KUKA KRL program: part3_2_post.src

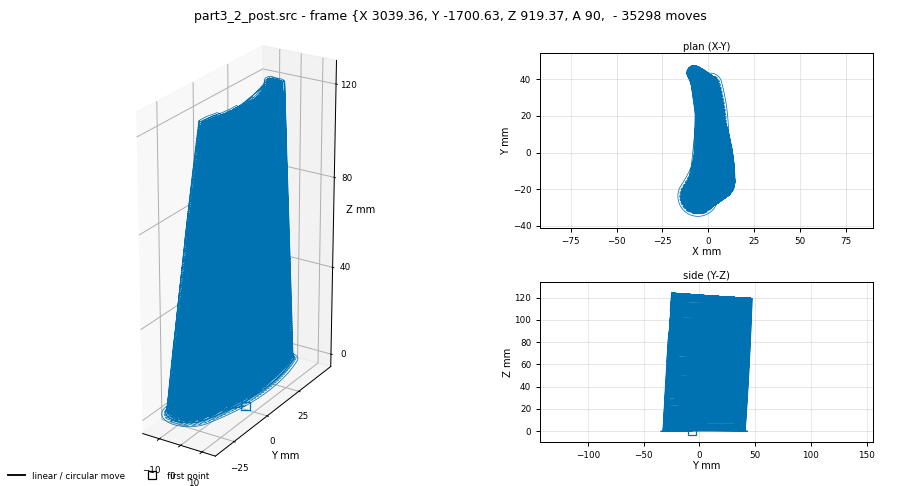
[picture p0: tool path of part3_2_post.src in frame {X 3039.36, Y -1700.63, Z 919.37, A 90, , 35298 of 35299 moves have a stored position in this frame; points joined in program order, loops and branches not executed]
&ACCESS RVO
&REL 3
DEF part3_2_post ( )

   ;---------------------RSI variable--------------------
   ; Declaration of KRL variables
   DECL INT ret	; Return value for RSI commands
   DECL INT CONTID	; ContainerID
   ;---------------------RSI variable--------------------

   ;---------------------RSI --------------------
   ret = RSI_CREATE("ros_rsi",CONTID,TRUE)
   IF (ret <> RSIOK) THEN
      HALT
   ENDIF

   ; Start RSI execution
   ret = RSI_ON(#ABSOLUTE)
   IF (ret <> RSIOK) THEN
      HALT
   ENDIF
   ;---------------------RSI--------------------

   ;FOLD INI
      ;FOLD BASISTECH INI
         GLOBAL INTERRUPT DECL 3 WHEN $STOPMESS==TRUE DO IR_STOPM ( )
         INTERRUPT ON 3
         BAS (#INITMOV,0 )
      ;ENDFOLD (BASISTECH INI)
      ;FOLD USER INI
         ;Make your modifications here

      ;ENDFOLD (USER INI)
   ;ENDFOLD (INI)

   $TOOL=TOOL_DATA[1] ; "LASER"
   ;$TOOL={X -5.25,Y -259.33,Z 286.75,A 0.0,B 0.0,C 0.0}
   $BASE={X 3039.36, Y -1700.63, Z 919.37, A 90, B 0, C 0}  ; user-defined BASE frame
   ;$BASE=BASE_DATA[3] ; user-defined BASE frame
   ;$BASE=BASE_DATA[1] ; "LK_BASE (TurnTable)"
   ;$BASE={X 1622.85,Y -1582.69,Z 15.62,A 0.14,B 0.07,C 0.25}

   $VEL.CP = 0.020 ; linear speed m/s
   $VEL.ORI1 = 300 ; swivel speed deg/s
   $VEL.ORI2 = 300 ; rotation speed deg/s

   $APO.CDIS = 0.3 ;mm; in ABB: zonddata = z0

   PTP $POS_ACT
   $OUT[15]=TRUE ; Wire touch signal bypass
   LaserOn_Ext()

   ;FOLD ANOUT ql_Power=0.1 ;%{PE}%R 8.5.19,%MKUKATPBASIS,%CANA,%VANOUT_STAT,%P 2:CHANNEL_1, 4:0.1
      $ANOUT[1]=0.179
   ;ENDFOLD

   LIN {X 9.999, Y -6.495, Z 0.000}
   LaserStart_Ext()
   LIN {X 9.851, Y -7.487, Z 0.000} C_DIS
   LIN {X 9.694, Y -8.478, Z 0.000} C_DIS
   LIN {X 9.517, Y -9.533, Z 0.000} C_DIS
   LIN {X 9.342, Y -10.520, Z 0.000} C_DIS
   LIN {X 9.158, Y -11.507, Z 0.000} C_DIS
   LIN {X 8.966, Y -12.491, Z 0.000} C_DIS
   LIN {X 8.778, Y -13.409, Z 0.000} C_DIS
   LIN {X 8.568, Y -14.390, Z 0.000} C_DIS
   LIN {X 8.350, Y -15.371, Z 0.000} C_DIS
   LIN {X 8.122, Y -16.349, Z 0.000} C_DIS
   LIN {X 7.886, Y -17.327, Z 0.000} C_DIS
   LIN {X 7.641, Y -18.302, Z 0.000} C_DIS
   LIN {X 7.387, Y -19.277, Z 0.000} C_DIS
   LIN {X 7.124, Y -20.250, Z 0.000} C_DIS
   LIN {X 6.851, Y -21.221, Z 0.000} C_DIS
   LIN {X 6.570, Y -22.190, Z 0.000} C_DIS
   LIN {X 6.300, Y -23.094, Z 0.000} C_DIS
   LIN {X 6.001, Y -24.061, Z 0.000} C_DIS
   LIN {X 5.693, Y -25.026, Z 0.000} C_DIS
   LIN {X 5.397, Y -25.926, Z 0.000} C_DIS
   LIN {X 5.181, Y -26.567, Z 0.000} C_DIS
   LIN {X 5.050, Y -26.952, Z 0.000} C_DIS
   LIN {X 4.961, Y -27.208, Z 0.000} C_DIS
   LIN {X 4.917, Y -27.337, Z 0.000} C_DIS
   LIN {X 4.841, Y -27.550, Z 0.000} C_DIS
   LIN {X 4.691, Y -27.934, Z 0.000} C_DIS
   LIN {X 4.448, Y -28.479, Z 0.000} C_DIS
   LIN {X 4.032, Y -29.267, Z 0.000} C_DIS
   LIN {X 3.511, Y -30.081, Z 0.000} C_DIS
   LIN {X 2.916, Y -30.853, Z 0.000} C_DIS
   LIN {X 2.255, Y -31.570, Z 0.000} C_DIS
   LIN {X 1.511, Y -32.247, Z 0.000} C_DIS
   LIN {X 0.738, Y -32.833, Z 0.000} C_DIS
   LIN {X -0.089, Y -33.352, Z 0.000} C_DIS
   LIN {X -0.956, Y -33.796, Z 0.000} C_DIS
   LIN {X -1.890, Y -34.172, Z 0.000} C_DIS
   LIN {X -2.855, Y -34.463, Z 0.000} C_DIS
   LIN {X -3.812, Y -34.661, Z 0.000} C_DIS
   LIN {X -4.777, Y -34.773, Z 0.000} C_DIS
   LIN {X -5.745, Y -34.799, Z 0.000} C_DIS
   LIN {X -6.715, Y -34.739, Z 0.000} C_DIS
   LIN {X -7.682, Y -34.593, Z 0.000} C_DIS
   LIN {X -8.661, Y -34.354, Z 0.000} C_DIS
   LIN {X -9.578, Y -34.041, Z 0.000} C_DIS
   LIN {X -10.468, Y -33.646, Z 0.000} C_DIS
   LIN {X -11.321, Y -33.170, Z 0.000} C_DIS
   LIN {X -12.123, Y -32.625, Z 0.000} C_DIS
   LIN {X -12.873, Y -32.012, Z 0.000} C_DIS
   LIN {X -13.571, Y -31.330, Z 0.000} C_DIS
   LIN {X -14.205, Y -30.589, Z 0.000} C_DIS
   LIN {X -14.787, Y -29.768, Z 0.000} C_DIS
   LIN {X -15.273, Y -28.929, Z 0.000} C_DIS
   LIN {X -15.686, Y -28.043, Z 0.000} C_DIS
   LIN {X -16.017, Y -27.128, Z 0.000} C_DIS
   LIN {X -16.282, Y -26.120, Z 0.000} C_DIS
   LIN {X -16.440, Y -25.161, Z 0.000} C_DIS
   LIN {X -16.513, Y -24.186, Z 0.000} C_DIS
   LIN {X -16.499, Y -23.215, Z 0.000} C_DIS
   LIN {X -16.400, Y -22.252, Z 0.000} C_DIS
   LIN {X -16.208, Y -21.260, Z 0.000} C_DIS
   LIN {X -15.937, Y -20.321, Z 0.000} C_DIS
   LIN {X -15.586, Y -19.416, Z 0.000} C_DIS
   LIN {X -15.139, Y -18.514, Z 0.000} C_DIS
   LIN {X -14.672, Y -17.743, Z 0.000} C_DIS
   LIN {X -14.112, Y -16.887, Z 0.000} C_DIS
   LIN {X -13.565, Y -16.024, Z 0.000} C_DIS
   LIN {X -13.060, Y -15.203, Z 0.000} C_DIS
   LIN {X -12.510, Y -14.277, Z 0.000} C_DIS
   LIN {X -12.002, Y -13.394, Z 0.000} C_DIS
   LIN {X -11.507, Y -12.503, Z 0.000} C_DIS
   LIN {X -11.025, Y -11.607, Z 0.000} C_DIS
   LIN {X -10.583, Y -10.753, Z 0.000} C_DIS
   LIN {X -10.126, Y -9.842, Z 0.000} C_DIS
   LIN {X -9.707, Y -8.975, Z 0.000} C_DIS
   LIN {X -9.276, Y -8.052, Z 0.000} C_DIS
   LIN {X -8.858, Y -7.124, Z 0.000} C_DIS
   LIN {X -8.455, Y -6.192, Z 0.000} C_DIS
   LIN {X -8.067, Y -5.258, Z 0.000} C_DIS
   LIN {X -7.693, Y -4.321, Z 0.000} C_DIS
   LIN {X -7.353, Y -3.432, Z 0.000} C_DIS
   LIN {X -6.987, Y -2.433, Z 0.000} C_DIS
   LIN {X -6.654, Y -1.483, Z 0.000} C_DIS
   LIN {X -6.352, Y -0.580, Z 0.000} C_DIS
   LIN {X -6.028, Y 0.435, Z 0.000} C_DIS
   LIN {X -5.735, Y 1.402, Z 0.000} C_DIS
   LIN {X -5.456, Y 2.373, Z 0.000} C_DIS
   LIN {X -5.163, Y 3.454, Z 0.000} C_DIS
   LIN {X -4.928, Y 4.375, Z 0.000} C_DIS
   LIN {X -4.693, Y 5.354, Z 0.000} C_DIS
   LIN {X -4.472, Y 6.338, Z 0.000} C_DIS
   LIN {X -4.264, Y 7.327, Z 0.000} C_DIS
   LIN {X -4.080, Y 8.268, Z 0.000} C_DIS
   LIN {X -3.900, Y 9.268, Z 0.000} C_DIS
   LIN {X -3.742, Y 10.214, Z 0.000} C_DIS
   LIN {X -3.582, Y 11.276, Z 0.000} C_DIS
   LIN {X -3.452, Y 12.228, Z 0.000} C_DIS
   LIN {X -3.328, Y 13.242, Z 0.000} C_DIS
   LIN {X -3.225, Y 14.200, Z 0.000} C_DIS
   LIN {X -3.130, Y 15.210, Z 0.000} C_DIS
   LIN {X -3.051, Y 16.218, Z 0.000} C_DIS
   LIN {X -2.988, Y 17.171, Z 0.000} C_DIS
   LIN {X -2.937, Y 18.180, Z 0.000} C_DIS
   LIN {X -2.899, Y 19.191, Z 0.000} C_DIS
   LIN {X -2.877, Y 20.145, Z 0.000} C_DIS
   LIN {X -2.868, Y 21.157, Z 0.000} C_DIS
   LIN {X -2.873, Y 22.168, Z 0.000} C_DIS
   LIN {X -2.891, Y 23.123, Z 0.000} C_DIS
   LIN {X -2.924, Y 24.133, Z 0.000} C_DIS
   LIN {X -2.971, Y 25.142, Z 0.000} C_DIS
   LIN {X -3.029, Y 26.094, Z 0.000} C_DIS
   LIN {X -3.104, Y 27.100, Z 0.000} C_DIS
   LIN {X -3.194, Y 28.106, Z 0.000} C_DIS
   LIN {X -3.291, Y 29.054, Z 0.000} C_DIS
   LIN {X -3.408, Y 30.058, Z 0.000} C_DIS
   LIN {X -3.540, Y 31.060, Z 0.000} C_DIS
   LIN {X -3.694, Y 32.116, Z 0.000} C_DIS
   LIN {X -3.855, Y 33.116, Z 0.000} C_DIS
   LIN {X -4.030, Y 34.115, Z 0.000} C_DIS
   LIN {X -4.219, Y 35.112, Z 0.000} C_DIS
   LIN {X -4.423, Y 36.108, Z 0.000} C_DIS
   LIN {X -4.573, Y 37.126, Z 0.000} C_DIS
   LIN {X -4.539, Y 38.127, Z 0.000} C_DIS
   LIN {X -4.338, Y 39.115, Z 0.000} C_DIS
   LIN {X -3.977, Y 40.053, Z 0.000} C_DIS
   LIN {X -3.442, Y 40.941, Z 0.000} C_DIS
   LIN {X -2.768, Y 41.711, Z 0.000} C_DIS
   LIN {X -1.943, Y 42.381, Z 0.000} C_DIS
   LIN {X -1.067, Y 42.875, Z 0.000} C_DIS
   LIN {X -0.126, Y 43.212, Z 0.000} C_DIS
   LIN {X 0.876, Y 43.381, Z 0.000} C_DIS
   LIN {X 1.877, Y 43.376, Z 0.000} C_DIS
   LIN {X 2.884, Y 43.202, Z 0.000} C_DIS
   LIN {X 3.835, Y 42.872, Z 0.000} C_DIS
   LIN {X 4.720, Y 42.387, Z 0.000} C_DIS
   LIN {X 5.506, Y 41.764, Z 0.000} C_DIS
   LIN {X 6.189, Y 41.003, Z 0.000} C_DIS
   LIN {X 6.758, Y 40.100, Z 0.000} C_DIS
   LIN {X 7.051, Y 39.435, Z 0.000} C_DIS
   LIN {X 7.216, Y 38.908, Z 0.000} C_DIS
   LIN {X 7.443, Y 38.057, Z 0.000} C_DIS
   LIN {X 7.697, Y 37.073, Z 0.000} C_DIS
   LIN {X 7.926, Y 36.154, Z 0.000} C_DIS
   LIN {X 8.177, Y 35.103, Z 0.000} C_DIS
   LIN {X 8.404, Y 34.115, Z 0.000} C_DIS
   LIN {X 8.621, Y 33.127, Z 0.000} C_DIS
   LIN {X 8.816, Y 32.203, Z 0.000} C_DIS
   LIN {X 9.042, Y 31.080, Z 0.000} C_DIS
   LIN {X 9.232, Y 30.088, Z 0.000} C_DIS
   LIN {X 9.413, Y 29.095, Z 0.000} C_DIS
   LIN {X 9.585, Y 28.100, Z 0.000} C_DIS
   LIN {X 9.738, Y 27.171, Z 0.000} C_DIS
   LIN {X 9.892, Y 26.174, Z 0.000} C_DIS
   LIN {X 10.038, Y 25.176, Z 0.000} C_DIS
   LIN {X 10.174, Y 24.176, Z 0.000} C_DIS
   LIN {X 10.294, Y 23.242, Z 0.000} C_DIS
   LIN {X 10.414, Y 22.241, Z 0.000} C_DIS
   LIN {X 10.531, Y 21.171, Z 0.000} C_DIS
   LIN {X 10.626, Y 20.234, Z 0.000} C_DIS
   LIN {X 10.718, Y 19.228, Z 0.000} C_DIS
   LIN {X 10.802, Y 18.222, Z 0.000} C_DIS
   LIN {X 10.872, Y 17.281, Z 0.000} C_DIS
   LIN {X 10.938, Y 16.273, Z 0.000} C_DIS
   LIN {X 10.995, Y 15.262, Z 0.000} C_DIS
   LIN {X 11.043, Y 14.251, Z 0.000} C_DIS
   LIN {X 11.080, Y 13.306, Z 0.000} C_DIS
   LIN {X 11.110, Y 12.292, Z 0.000} C_DIS
   LIN {X 11.131, Y 11.277, Z 0.000} C_DIS
   LIN {X 11.143, Y 10.328, Z 0.000} C_DIS
   LIN {X 11.146, Y 9.313, Z 0.000} C_DIS
   LIN {X 11.141, Y 8.365, Z 0.000} C_DIS
   LIN {X 11.126, Y 7.350, Z 0.000} C_DIS
   LIN {X 11.103, Y 6.336, Z 0.000} C_DIS
   LIN {X 11.070, Y 5.325, Z 0.000} C_DIS
   LIN {X 11.031, Y 4.382, Z 0.000} C_DIS
   LIN {X 10.980, Y 3.374, Z 0.000} C_DIS
   LIN {X 10.921, Y 2.367, Z 0.000} C_DIS
   LIN {X 10.852, Y 1.361, Z 0.000} C_DIS
   LIN {X 10.774, Y 0.358, Z 0.000} C_DIS
   LIN {X 10.694, Y -0.578, Z 0.000} C_DIS
   LIN {X 10.599, Y -1.579, Z 0.000} C_DIS
   LIN {X 10.495, Y -2.578, Z 0.000} C_DIS
   LIN {X 10.382, Y -3.576, Z 0.000} C_DIS
   LIN {X 10.260, Y -4.573, Z 0.000} C_DIS
   LIN {X 10.138, Y -5.502, Z 0.000} C_DIS
   LIN {X 9.999, Y -6.495, Z 0.000}
   LaserEnd_Ext()
   LIN {X -8.478, Y -33.360, Z 0.000}
   LaserStart_Ext()
   LIN {X -2.661, Y -33.360, Z 0.000}
   LaserEnd_Ext()
   LIN {X -0.389, Y -32.360, Z 0.000}
   LaserStart_Ext()
   LIN {X -10.721, Y -32.360, Z 0.000}
   LaserEnd_Ext()
   LIN {X -12.090, Y -31.360, Z 0.000}
   LaserStart_Ext()
   LIN {X 1.000, Y -31.360, Z 0.000}
   LaserEnd_Ext()
   LIN {X 2.010, Y -30.360, Z 0.000}
   LaserStart_Ext()
   LIN {X -13.085, Y -30.360, Z 0.000}
   LaserEnd_Ext()
   LIN {X -13.850, Y -29.360, Z 0.000}
   LaserStart_Ext()
   LIN {X 2.785, Y -29.360, Z 0.000}
   LaserEnd_Ext()
   LIN {X 3.380, Y -28.360, Z 0.000}
   LaserStart_Ext()
   LIN {X -14.435, Y -28.360, Z 0.000}
   LaserEnd_Ext()
   LIN {X -14.870, Y -27.360, Z 0.000}
   LaserStart_Ext()
   LIN {X 3.841, Y -27.360, Z 0.000}
   LaserEnd_Ext()
   LIN {X 4.196, Y -26.360, Z 0.000}
   LaserStart_Ext()
   LIN {X -15.185, Y -26.360, Z 0.000}
   LaserEnd_Ext()
   LIN {X -15.394, Y -25.360, Z 0.000}
   LaserStart_Ext()
   LIN {X 4.531, Y -25.360, Z 0.000}
   LaserEnd_Ext()
   LIN {X 4.856, Y -24.360, Z 0.000}
   LaserStart_Ext()
   LIN {X -15.497, Y -24.360, Z 0.000}
   LaserEnd_Ext()
   LIN {X -15.501, Y -23.360, Z 0.000}
   LaserStart_Ext()
   LIN {X 5.171, Y -23.360, Z 0.000}
   LaserEnd_Ext()
   LIN {X 5.475, Y -22.360, Z 0.000}
   LaserStart_Ext()
   LIN {X -15.403, Y -22.360, Z 0.000}
   LaserEnd_Ext()
   LIN {X -15.196, Y -21.360, Z 0.000}
   LaserStart_Ext()
   LIN {X 5.770, Y -21.360, Z 0.000}
   LaserEnd_Ext()
   LIN {X 6.054, Y -20.360, Z 0.000}
   LaserStart_Ext()
   LIN {X -14.879, Y -20.360, Z 0.000}
   LaserEnd_Ext()
   LIN {X -14.442, Y -19.360, Z 0.000}
   LaserStart_Ext()
   LIN {X 6.328, Y -19.360, Z 0.000}
   LaserEnd_Ext()
   LIN {X 6.592, Y -18.360, Z 0.000}
   LaserStart_Ext()
   LIN {X -13.876, Y -18.360, Z 0.000}
   LaserEnd_Ext()
   LIN {X -13.228, Y -17.360, Z 0.000}
   LaserStart_Ext()
   LIN {X 6.847, Y -17.360, Z 0.000}
   LaserEnd_Ext()
   LIN {X 7.091, Y -16.360, Z 0.000}
   LaserStart_Ext()
   LIN {X -12.598, Y -16.360, Z 0.000}
   LaserEnd_Ext()
   LIN {X -11.990, Y -15.360, Z 0.000}
   LaserStart_Ext()
   LIN {X 7.326, Y -15.360, Z 0.000}
   LaserEnd_Ext()
   LIN {X 7.551, Y -14.360, Z 0.000}
   LaserStart_Ext()
   LIN {X -11.404, Y -14.360, Z 0.000}
   LaserEnd_Ext()
   LIN {X -10.839, Y -13.360, Z 0.000}
   LaserStart_Ext()
   LIN {X 7.766, Y -13.360, Z 0.000}
   LaserEnd_Ext()
   LIN {X 7.972, Y -12.360, Z 0.000}
   LaserStart_Ext()
   LIN {X -10.295, Y -12.360, Z 0.000}
   LaserEnd_Ext()
   LIN {X -9.771, Y -11.360, Z 0.000}
   LaserStart_Ext()
   LIN {X 8.168, Y -11.360, Z 0.000}
   LaserEnd_Ext()
   LIN {X 8.355, Y -10.360, Z 0.000}
   LaserStart_Ext()
   LIN {X -9.267, Y -10.360, Z 0.000}
   LaserEnd_Ext()
   LIN {X -8.783, Y -9.360, Z 0.000}
   LaserStart_Ext()
   LIN {X 8.532, Y -9.360, Z 0.000}
   LaserEnd_Ext()
   LIN {X 8.700, Y -8.360, Z 0.000}
   LaserStart_Ext()
   LIN {X -8.318, Y -8.360, Z 0.000}
   LaserEnd_Ext()
   LIN {X -7.871, Y -7.360, Z 0.000}
   LaserStart_Ext()
   LIN {X 8.859, Y -7.360, Z 0.000}
   LaserEnd_Ext()
   LIN {X 9.008, Y -6.360, Z 0.000}
   LaserStart_Ext()
   LIN {X -7.442, Y -6.360, Z 0.000}
   LaserEnd_Ext()
   LIN {X -7.031, Y -5.360, Z 0.000}
   LaserStart_Ext()
   LIN {X 9.148, Y -5.360, Z 0.000}
   LaserEnd_Ext()
   LIN {X 9.278, Y -4.360, Z 0.000}
   LaserStart_Ext()
   LIN {X -6.638, Y -4.360, Z 0.000}
   LaserEnd_Ext()
   LIN {X -6.261, Y -3.360, Z 0.000}
   LaserStart_Ext()
   LIN {X 9.400, Y -3.360, Z 0.000}
   LaserEnd_Ext()
   LIN {X 9.512, Y -2.360, Z 0.000}
   LaserStart_Ext()
   LIN {X -5.902, Y -2.360, Z 0.000}
   LaserEnd_Ext()
   LIN {X -5.558, Y -1.360, Z 0.000}
   LaserStart_Ext()
   LIN {X 9.615, Y -1.360, Z 0.000}
   LaserEnd_Ext()
   LIN {X 9.709, Y -0.360, Z 0.000}
   LaserStart_Ext()
   LIN {X -5.232, Y -0.360, Z 0.000}
   LaserEnd_Ext()
   LIN {X -4.921, Y 0.640, Z 0.000}
   LaserStart_Ext()
   LIN {X 9.793, Y 0.640, Z 0.000}
   LaserEnd_Ext()
   LIN {X 9.869, Y 1.640, Z 0.000}
   LaserStart_Ext()
   LIN {X -4.627, Y 1.640, Z 0.000}
   LaserEnd_Ext()
   LIN {X -4.348, Y 2.640, Z 0.000}
   LaserStart_Ext()
   LIN {X 9.935, Y 2.640, Z 0.000}
   LaserEnd_Ext()
   LIN {X 9.992, Y 3.640, Z 0.000}
   LaserStart_Ext()
   LIN {X -4.084, Y 3.640, Z 0.000}
   LaserEnd_Ext()
   LIN {X -3.836, Y 4.640, Z 0.000}
   LaserStart_Ext()
   LIN {X 10.041, Y 4.640, Z 0.000}
   LaserEnd_Ext()
   LIN {X 10.080, Y 5.640, Z 0.000}
   LaserStart_Ext()
   LIN {X -3.604, Y 5.640, Z 0.000}
   LaserEnd_Ext()
   LIN {X -3.387, Y 6.640, Z 0.000}
   LaserStart_Ext()
   LIN {X 10.110, Y 6.640, Z 0.000}
   LaserEnd_Ext()
   LIN {X 10.130, Y 7.640, Z 0.000}
   LaserStart_Ext()
   LIN {X -3.184, Y 7.640, Z 0.000}
   LaserEnd_Ext()
   LIN {X -2.997, Y 8.640, Z 0.000}
   LaserStart_Ext()
   LIN {X 10.142, Y 8.640, Z 0.000}
   LaserEnd_Ext()
   LIN {X 10.145, Y 9.640, Z 0.000}
   LaserStart_Ext()
   LIN {X -2.824, Y 9.640, Z 0.000}
   LaserEnd_Ext()
   LIN {X -2.667, Y 10.640, Z 0.000}
   LaserStart_Ext()
   LIN {X 10.139, Y 10.640, Z 0.000}
   LaserEnd_Ext()
   LIN {X 10.123, Y 11.640, Z 0.000}
   LaserStart_Ext()
   LIN {X -2.523, Y 11.640, Z 0.000}
   LaserEnd_Ext()
   LIN {X -2.394, Y 12.640, Z 0.000}
   LaserStart_Ext()
   LIN {X 10.099, Y 12.640, Z 0.000}
   LaserEnd_Ext()
   LIN {X 10.066, Y 13.640, Z 0.000}
   LaserStart_Ext()
   LIN {X -2.280, Y 13.640, Z 0.000}
   LaserEnd_Ext()
   LIN {X -2.179, Y 14.640, Z 0.000}
   LaserStart_Ext()
   LIN {X 10.024, Y 14.640, Z 0.000}
   LaserEnd_Ext()
   LIN {X 9.972, Y 15.640, Z 0.000}
   LaserStart_Ext()
   LIN {X -2.093, Y 15.640, Z 0.000}
   LaserEnd_Ext()
   LIN {X -2.021, Y 16.640, Z 0.000}
   LaserStart_Ext()
   LIN {X 9.912, Y 16.640, Z 0.000}
   LaserEnd_Ext()
   LIN {X 9.842, Y 17.640, Z 0.000}
   LaserStart_Ext()
   LIN {X -1.963, Y 17.640, Z 0.000}
   LaserEnd_Ext()
   LIN {X -1.919, Y 18.640, Z 0.000}
   LaserStart_Ext()
   LIN {X 9.764, Y 18.640, Z 0.000}
   LaserEnd_Ext()
   LIN {X 9.676, Y 19.640, Z 0.000}
   LaserStart_Ext()
   LIN {X -1.889, Y 19.640, Z 0.000}
   LaserEnd_Ext()
   LIN {X -1.873, Y 20.640, Z 0.000}
   LaserStart_Ext()
   LIN {X 9.580, Y 20.640, Z 0.000}
   LaserEnd_Ext()
   LIN {X 9.474, Y 21.640, Z 0.000}
   LaserStart_Ext()
   LIN {X -1.871, Y 21.640, Z 0.000}
   LaserEnd_Ext()
   LIN {X -1.882, Y 22.640, Z 0.000}
   LaserStart_Ext()
   LIN {X 9.359, Y 22.640, Z 0.000}
   LaserEnd_Ext()
   LIN {X 9.235, Y 23.640, Z 0.000}
   LaserStart_Ext()
   LIN {X -1.908, Y 23.640, Z 0.000}
   LaserEnd_Ext()
   LIN {X -1.947, Y 24.640, Z 0.000}
   LaserStart_Ext()
   LIN {X 9.102, Y 24.640, Z 0.000}
   LaserEnd_Ext()
   LIN {X 8.959, Y 25.640, Z 0.000}
   LaserStart_Ext()
   LIN {X -2.000, Y 25.640, Z 0.000}
   LaserEnd_Ext()
   LIN {X -2.067, Y 26.640, Z 0.000}
   LaserStart_Ext()
   LIN {X 8.808, Y 26.640, Z 0.000}
   LaserEnd_Ext()
   LIN {X 8.647, Y 27.640, Z 0.000}
   LaserStart_Ext()
   LIN {X -2.148, Y 27.640, Z 0.000}
   LaserEnd_Ext()
   LIN {X -2.243, Y 28.640, Z 0.000}
   LaserStart_Ext()
   LIN {X 8.477, Y 28.640, Z 0.000}
   LaserEnd_Ext()
   LIN {X 8.297, Y 29.640, Z 0.000}
   LaserStart_Ext()
   LIN {X -2.353, Y 29.640, Z 0.000}
   LaserEnd_Ext()
   LIN {X -2.476, Y 30.640, Z 0.000}
   LaserStart_Ext()
   LIN {X 8.109, Y 30.640, Z 0.000}
   LaserEnd_Ext()
   LIN {X 7.910, Y 31.640, Z 0.000}
   LaserStart_Ext()
   LIN {X -2.614, Y 31.640, Z 0.000}
   LaserEnd_Ext()
   LIN {X -2.765, Y 32.640, Z 0.000}
   LaserStart_Ext()
   LIN {X 7.702, Y 32.640, Z 0.000}
   LaserEnd_Ext()
   LIN {X 7.485, Y 33.640, Z 0.000}
   LaserStart_Ext()
   LIN {X -2.931, Y 33.640, Z 0.000}
   LaserEnd_Ext()
   LIN {X -3.111, Y 34.640, Z 0.000}
   LaserStart_Ext()
   LIN {X 7.258, Y 34.640, Z 0.000}
   LaserEnd_Ext()
   LIN {X 7.020, Y 35.640, Z 0.000}
   LaserStart_Ext()
   LIN {X -3.306, Y 35.640, Z 0.000}
   LaserEnd_Ext()
   LIN {X -3.490, Y 36.640, Z 0.000}
   LaserStart_Ext()
   LIN {X 6.774, Y 36.640, Z 0.000}
   LaserEnd_Ext()
   LIN {X 6.518, Y 37.640, Z 0.000}
   LaserStart_Ext()
   LIN {X -3.555, Y 37.640, Z 0.000}
   LaserEnd_Ext()
   LIN {X -3.414, Y 38.640, Z 0.000}
   LaserStart_Ext()
   LIN {X 6.252, Y 38.640, Z 0.000}
   LaserEnd_Ext()
   LIN {X 5.866, Y 39.640, Z 0.000}
   LaserStart_Ext()
   LIN {X -3.059, Y 39.640, Z 0.000}
   LaserEnd_Ext()
   LIN {X -2.377, Y 40.640, Z 0.000}
   LaserStart_Ext()
   LIN {X 5.172, Y 40.640, Z 0.000}
   LaserEnd_Ext()
   LIN {X 4.003, Y 41.640, Z 0.000}
   LaserStart_Ext()
   LIN {X -1.221, Y 41.640, Z 0.000}
   LaserEnd_Ext()
   LIN {X 8.972, Y -2.779, Z 0.850}
   LaserStart_Ext()
   LIN {X 8.898, Y -3.428, Z 0.850} C_DIS
   LIN {X 8.854, Y -3.793, Z 0.850} C_DIS
   LIN {X 8.778, Y -4.409, Z 0.850} C_DIS
   LIN {X 8.735, Y -4.751, Z 0.850} C_DIS
   LIN {X 8.652, Y -5.371, Z 0.850} C_DIS
   LIN {X 8.602, Y -5.739, Z 0.850} C_DIS
   LIN {X 8.513, Y -6.364, Z 0.850} C_DIS
   LIN {X 8.459, Y -6.734, Z 0.850} C_DIS
   LIN {X 8.370, Y -7.324, Z 0.850} C_DIS
   LIN {X 8.313, Y -7.695, Z 0.850} C_DIS
   LIN {X 8.211, Y -8.329, Z 0.850} C_DIS
   LIN {X 8.146, Y -8.726, Z 0.850} C_DIS
   LIN {X 8.044, Y -9.325, Z 0.850} C_DIS
   LIN {X 7.979, Y -9.698, Z 0.850} C_DIS
   LIN {X 7.864, Y -10.341, Z 0.850} C_DIS
   LIN {X 7.795, Y -10.716, Z 0.850} C_DIS
   LIN {X 7.681, Y -11.322, Z 0.850} C_DIS
   LIN {X 7.609, Y -11.698, Z 0.850} C_DIS
   LIN {X 7.538, Y -12.049, Z 0.850} C_DIS
   LIN {X 7.409, Y -12.700, Z 0.850} C_DIS
   LIN {X 7.330, Y -13.078, Z 0.850} C_DIS
   LIN {X 7.210, Y -13.651, Z 0.850} C_DIS
   LIN {X 7.127, Y -14.029, Z 0.850} C_DIS
   LIN {X 6.993, Y -14.647, Z 0.850} C_DIS
   LIN {X 6.906, Y -15.027, Z 0.850} C_DIS
   LIN {X 6.774, Y -15.606, Z 0.850} C_DIS
   LIN {X 6.684, Y -15.987, Z 0.850} C_DIS
   LIN {X 6.536, Y -16.610, Z 0.850} C_DIS
   LIN {X 6.297, Y -17.577, Z 0.850} C_DIS
   LIN {X 6.199, Y -17.959, Z 0.850} C_DIS
   LIN {X 6.048, Y -18.547, Z 0.850} C_DIS
   LIN {X 5.946, Y -18.930, Z 0.850} C_DIS
   LIN {X 5.788, Y -19.520, Z 0.850} C_DIS
   LIN {X 5.682, Y -19.905, Z 0.850} C_DIS
   LIN {X 5.519, Y -20.497, Z 0.850} C_DIS
   LIN {X 5.409, Y -20.882, Z 0.850} C_DIS
   LIN {X 5.250, Y -21.434, Z 0.850} C_DIS
   LIN {X 5.144, Y -21.794, Z 0.850} C_DIS
   LIN {X 4.968, Y -22.391, Z 0.850} C_DIS
   LIN {X 4.850, Y -22.778, Z 0.850} C_DIS
   LIN {X 4.680, Y -23.333, Z 0.850} C_DIS
   LIN {X 4.558, Y -23.721, Z 0.850} C_DIS
   LIN {X 4.382, Y -24.278, Z 0.850} C_DIS
   LIN {X 4.264, Y -24.641, Z 0.850} C_DIS
   LIN {X 4.068, Y -25.243, Z 0.850} C_DIS
   LIN {X 3.908, Y -25.429, Z 0.850} C_DIS
   LIN {X 3.630, Y -26.087, Z 0.850} C_DIS
   LIN {X 3.542, Y -26.333, Z 0.850} C_DIS
   LIN {X 3.423, Y -26.817, Z 0.850} C_DIS
   LIN {X 3.209, Y -27.251, Z 0.850} C_DIS
   LIN {X 3.097, Y -27.514, Z 0.850} C_DIS
   LIN {X 2.678, Y -28.454, Z 0.850} C_DIS
   LIN {X 2.399, Y -28.904, Z 0.850} C_DIS
   LIN {X 2.097, Y -29.342, Z 0.850} C_DIS
   LIN {X 1.765, Y -29.763, Z 0.850} C_DIS
   LIN {X 1.431, Y -30.148, Z 0.850} C_DIS
   LIN {X 1.051, Y -30.534, Z 0.850} C_DIS
   LIN {X 0.696, Y -30.863, Z 0.850} C_DIS
   LIN {X 0.278, Y -31.206, Z 0.850} C_DIS
   LIN {X -0.091, Y -31.481, Z 0.850} C_DIS
   LIN {X -0.574, Y -31.797, Z 0.850} C_DIS
   LIN {X -0.969, Y -32.030, Z 0.850} C_DIS
   LIN {X -1.500, Y -32.298, Z 0.850} C_DIS
   LIN {X -1.804, Y -32.465, Z 0.850} C_DIS
   LIN {X -2.420, Y -32.697, Z 0.850} C_DIS
   LIN {X -2.707, Y -32.892, Z 0.850} C_DIS
   LIN {X -3.468, Y -33.085, Z 0.850} C_DIS
   LIN {X -3.681, Y -33.136, Z 0.850} C_DIS
   LIN {X -3.853, Y -33.058, Z 0.850} C_DIS
   LIN {X -4.484, Y -33.150, Z 0.850} C_DIS
   LIN {X -4.819, Y -33.216, Z 0.850} C_DIS
   LIN {X -5.534, Y -33.241, Z 0.850} C_DIS
   LIN {X -5.833, Y -33.304, Z 0.850} C_DIS
   LIN {X -6.626, Y -33.243, Z 0.850} C_DIS
   LIN {X -6.821, Y -33.219, Z 0.850} C_DIS
   LIN {X -7.621, Y -33.069, Z 0.850} C_DIS
   LIN {X -7.812, Y -33.028, Z 0.850} C_DIS
   LIN {X -7.896, Y -32.915, Z 0.850} C_DIS
   LIN {X -8.565, Y -32.715, Z 0.850} C_DIS
   LIN {X -8.863, Y -32.639, Z 0.850} C_DIS
   LIN {X -9.586, Y -32.332, Z 0.850} C_DIS
   LIN {X -9.840, Y -32.267, Z 0.850} C_DIS
   LIN {X -10.556, Y -31.862, Z 0.850} C_DIS
   LIN {X -10.699, Y -31.771, Z 0.850} C_DIS
   LIN {X -11.372, Y -31.287, Z 0.850} C_DIS
   LIN {X -11.503, Y -31.185, Z 0.850} C_DIS
   LIN {X -12.135, Y -30.617, Z 0.850} C_DIS
   LIN {X -12.256, Y -30.505, Z 0.850} C_DIS
   LIN {X -12.366, Y -30.383, Z 0.850} C_DIS
   LIN {X -12.926, Y -29.756, Z 0.850} C_DIS
   LIN {X -13.026, Y -29.622, Z 0.850} C_DIS
   LIN {X -13.523, Y -28.921, Z 0.850} C_DIS
   LIN {X -13.607, Y -28.784, Z 0.850} C_DIS
   LIN {X -14.009, Y -28.056, Z 0.850} C_DIS
   LIN {X -14.081, Y -27.911, Z 0.850} C_DIS
   LIN {X -14.051, Y -27.799, Z 0.850} C_DIS
   LIN {X -14.340, Y -27.107, Z 0.850} C_DIS
   LIN {X -14.459, Y -26.847, Z 0.850} C_DIS
   LIN {X -14.684, Y -26.082, Z 0.850} C_DIS
   LIN {X -14.782, Y -25.852, Z 0.850} C_DIS
   LIN {X -14.932, Y -25.020, Z 0.850} C_DIS
   LIN {X -14.949, Y -24.850, Z 0.850} C_DIS
   LIN {X -15.005, Y -24.032, Z 0.850} C_DIS
   LIN {X -15.007, Y -23.856, Z 0.850} C_DIS
   LIN {X -14.975, Y -23.053, Z 0.850} C_DIS
   LIN {X -14.961, Y -22.872, Z 0.850} C_DIS
   LIN {X -14.839, Y -22.055, Z 0.850} C_DIS
   LIN {X -14.681, Y -21.717, Z 0.850} C_DIS
   LIN {X -14.505, Y -21.059, Z 0.850} C_DIS
   LIN {X -14.419, Y -20.793, Z 0.850} C_DIS
   LIN {X -14.179, Y -20.172, Z 0.850} C_DIS
   LIN {X -14.094, Y -19.902, Z 0.850} C_DIS
   LIN {X -13.922, Y -19.670, Z 0.850} C_DIS
   LIN {X -13.450, Y -18.845, Z 0.850} C_DIS
   LIN {X -13.347, Y -18.620, Z 0.850} C_DIS
   LIN {X -13.053, Y -18.146, Z 0.850} C_DIS
   LIN {X -12.875, Y -17.854, Z 0.850} C_DIS
   LIN {X -12.581, Y -17.359, Z 0.850} C_DIS
   LIN {X -12.047, Y -16.505, Z 0.850} C_DIS
   LIN {X -11.665, Y -15.874, Z 0.850} C_DIS
   LIN {X -11.514, Y -15.624, Z 0.850} C_DIS
   LIN {X -11.156, Y -15.015, Z 0.850} C_DIS
   LIN {X -11.016, Y -14.775, Z 0.850} C_DIS
   LIN {X -10.643, Y -14.120, Z 0.850} C_DIS
   LIN {X -10.505, Y -13.876, Z 0.850} C_DIS
   LIN {X -10.152, Y -13.235, Z 0.850} C_DIS
   LIN {X -10.017, Y -12.988, Z 0.850} C_DIS
   LIN {X -9.672, Y -12.339, Z 0.850} C_DIS
   LIN {X -9.547, Y -12.102, Z 0.850} C_DIS
   LIN {X -9.212, Y -11.450, Z 0.850} C_DIS
   LIN {X -9.081, Y -11.195, Z 0.850} C_DIS
   LIN {X -8.759, Y -10.546, Z 0.850} C_DIS
   LIN {X -8.638, Y -10.301, Z 0.850} C_DIS
   LIN {X -8.330, Y -9.659, Z 0.850} C_DIS
   LIN {X -8.205, Y -9.396, Z 0.850} C_DIS
   LIN {X -7.912, Y -8.765, Z 0.850} C_DIS
   LIN {X -7.790, Y -8.498, Z 0.850} C_DIS
   LIN {X -7.497, Y -7.843, Z 0.850} C_DIS
   LIN {X -7.378, Y -7.573, Z 0.850} C_DIS
   LIN {X -7.103, Y -6.933, Z 0.850} C_DIS
   LIN {X -6.987, Y -6.661, Z 0.850} C_DIS
   LIN {X -6.713, Y -5.999, Z 0.850} C_DIS
   LIN {X -6.601, Y -5.724, Z 0.850} C_DIS
   LIN {X -6.329, Y -5.041, Z 0.850} C_DIS
   LIN {X -6.226, Y -4.777, Z 0.850} C_DIS
   LIN {X -5.974, Y -4.118, Z 0.850} C_DIS
   LIN {X -5.862, Y -3.820, Z 0.850} C_DIS
   LIN {X -5.631, Y -3.188, Z 0.850} C_DIS
   LIN {X -5.528, Y -2.901, Z 0.850} C_DIS
   LIN {X -5.300, Y -2.253, Z 0.850} C_DIS
   LIN {X -5.206, Y -1.979, Z 0.850} C_DIS
   LIN {X -4.983, Y -1.315, Z 0.850} C_DIS
   LIN {X -4.881, Y -1.004, Z 0.850} C_DIS
   LIN {X -4.663, Y -0.324, Z 0.850} C_DIS
   LIN {X -4.571, Y -0.025, Z 0.850} C_DIS
   LIN {X -4.373, Y 0.620, Z 0.850} C_DIS
   LIN {X -4.284, Y 0.922, Z 0.850} C_DIS
   LIN {X -4.093, Y 1.581, Z 0.850} C_DIS
   LIN {X -3.998, Y 1.920, Z 0.850} C_DIS
   LIN {X -3.813, Y 2.593, Z 0.850} C_DIS
   LIN {X -3.736, Y 2.884, Z 0.850} C_DIS
   LIN {X -3.557, Y 3.571, Z 0.850} C_DIS
   LIN {X -3.480, Y 3.883, Z 0.850} C_DIS
   LIN {X -3.322, Y 4.527, Z 0.850} C_DIS
   LIN {X -3.248, Y 4.843, Z 0.850} C_DIS
   LIN {X -3.085, Y 5.549, Z 0.850} C_DIS
   LIN {X -3.015, Y 5.870, Z 0.850} C_DIS
   LIN {X -2.870, Y 6.543, Z 0.850} C_DIS
   LIN {X -2.808, Y 6.850, Z 0.850} C_DIS
   LIN {X -2.679, Y 7.489, Z 0.850} C_DIS
   LIN {X -2.617, Y 7.818, Z 0.850} C_DIS
   LIN {X -2.493, Y 8.484, Z 0.850} C_DIS
   LIN {X -2.438, Y 8.797, Z 0.850} C_DIS
   LIN {X -2.320, Y 9.483, Z 0.850} C_DIS
   LIN {X -2.217, Y 10.137, Z 0.850} C_DIS
   LIN {X -2.161, Y 10.493, Z 0.850} C_DIS
   LIN {X -2.066, Y 11.155, Z 0.850} C_DIS
   LIN {X -2.019, Y 11.477, Z 0.850} C_DIS
   LIN {X -1.935, Y 12.129, Z 0.850} C_DIS
   LIN {X -1.890, Y 12.474, Z 0.850} C_DIS
   LIN {X -1.816, Y 13.113, Z 0.850} C_DIS
   LIN {X -1.778, Y 13.442, Z 0.850} C_DIS
   LIN {X -1.710, Y 14.117, Z 0.850} C_DIS
   LIN {X -1.674, Y 14.466, Z 0.850} C_DIS
   LIN {X -1.616, Y 15.130, Z 0.850} C_DIS
   LIN {X -1.586, Y 15.481, Z 0.850} C_DIS
   LIN {X -1.538, Y 16.134, Z 0.850} C_DIS
   LIN {X -1.514, Y 16.468, Z 0.850} C_DIS
   LIN {X -1.475, Y 17.111, Z 0.850} C_DIS
   LIN {X -1.454, Y 17.467, Z 0.850} C_DIS
   LIN {X -1.425, Y 18.098, Z 0.850} C_DIS
   LIN {X -1.409, Y 18.457, Z 0.850} C_DIS
   LIN {X -1.388, Y 19.119, Z 0.850} C_DIS
   LIN {X -1.378, Y 19.460, Z 0.850} C_DIS
   LIN {X -1.366, Y 20.109, Z 0.850} C_DIS
   LIN {X -1.360, Y 20.472, Z 0.850} C_DIS
   LIN {X -1.357, Y 21.109, Z 0.850} C_DIS
   LIN {X -1.356, Y 21.475, Z 0.850} C_DIS
   LIN {X -1.361, Y 22.100, Z 0.850} C_DIS
   LIN {X -1.365, Y 22.447, Z 0.850} C_DIS
   LIN {X -1.380, Y 23.097, Z 0.850} C_DIS
   LIN {X -1.389, Y 23.467, Z 0.850} C_DIS
   LIN {X -1.412, Y 24.102, Z 0.850} C_DIS
   LIN {X -1.427, Y 24.474, Z 0.850} C_DIS
   LIN {X -1.460, Y 25.131, Z 0.850} C_DIS
   LIN {X -1.479, Y 25.484, Z 0.850} C_DIS
   LIN {X -1.518, Y 26.091, Z 0.850} C_DIS
   LIN {X -1.543, Y 26.466, Z 0.850} C_DIS
   LIN {X -1.592, Y 27.093, Z 0.850} C_DIS
   LIN {X -1.622, Y 27.470, Z 0.850} C_DIS
   LIN {X -1.681, Y 28.115, Z 0.850} C_DIS
   LIN {X -1.715, Y 28.473, Z 0.850} C_DIS
   LIN {X -1.782, Y 29.100, Z 0.850} C_DIS
   LIN {X -1.823, Y 29.481, Z 0.850} C_DIS
   LIN {X -1.897, Y 30.090, Z 0.850} C_DIS
   LIN {X -1.944, Y 30.473, Z 0.850} C_DIS
   LIN {X -2.027, Y 31.097, Z 0.850} C_DIS
   LIN {X -2.084, Y 31.503, Z 0.850} C_DIS
   LIN {X -2.173, Y 32.108, Z 0.850} C_DIS
   LIN {X -2.232, Y 32.494, Z 0.850} C_DIS
   LIN {X -2.332, Y 33.109, Z 0.850} C_DIS
   LIN {X -2.397, Y 33.497, Z 0.850} C_DIS
   LIN {X -2.507, Y 34.120, Z 0.850} C_DIS
   LIN {X -2.578, Y 34.510, Z 0.850} C_DIS
   LIN {X -2.697, Y 35.382, Z 0.850} C_DIS
   LIN {X -2.747, Y 35.588, Z 0.850} C_DIS
   LIN {X -2.775, Y 36.128, Z 0.850} C_DIS
   LIN {X -2.870, Y 36.493, Z 0.850} C_DIS
   LIN {X -2.884, Y 36.786, Z 0.850} C_DIS
   LIN {X -3.034, Y 37.435, Z 0.850} C_DIS
   LIN {X -3.056, Y 38.001, Z 0.850} C_DIS
   LIN {X -2.993, Y 38.437, Z 0.850} C_DIS
   LIN {X -2.893, Y 38.777, Z 0.850} C_DIS
   LIN {X -2.682, Y 39.334, Z 0.850} C_DIS
   LIN {X -2.520, Y 39.663, Z 0.850} C_DIS
   LIN {X -2.304, Y 39.957, Z 0.850} C_DIS
   LIN {X -1.373, Y 40.852, Z 0.850} C_DIS
   LIN {X -1.236, Y 40.945, Z 0.850} C_DIS
   LIN {X -0.535, Y 41.382, Z 0.850} C_DIS
   LIN {X -0.396, Y 41.446, Z 0.850} C_DIS
   LIN {X -0.248, Y 41.485, Z 0.850} C_DIS
   LIN {X 0.585, Y 41.747, Z 0.850} C_DIS
   LIN {X 1.533, Y 41.785, Z 0.850} C_DIS
   LIN {X 1.754, Y 41.785, Z 0.850} C_DIS
   LIN {X 2.713, Y 41.577, Z 0.850} C_DIS
   LIN {X 2.864, Y 41.525, Z 0.850} C_DIS
   LIN {X 3.717, Y 41.107, Z 0.850} C_DIS
   LIN {X 4.533, Y 40.430, Z 0.850} C_DIS
   LIN {X 4.687, Y 40.222, Z 0.850} C_DIS
   LIN {X 5.213, Y 39.535, Z 0.850} C_DIS
   LIN {X 5.651, Y 38.504, Z 0.850} C_DIS
   LIN {X 5.697, Y 38.269, Z 0.850} C_DIS
   LIN {X 5.864, Y 37.799, Z 0.850} C_DIS
   LIN {X 6.100, Y 37.156, Z 0.850} C_DIS
   LIN {X 6.164, Y 36.904, Z 0.850} C_DIS
   LIN {X 6.342, Y 36.206, Z 0.850} C_DIS
   LIN {X 6.412, Y 35.915, Z 0.850} C_DIS
   LIN {X 6.585, Y 35.210, Z 0.850} C_DIS
   LIN {X 6.650, Y 34.934, Z 0.850} C_DIS
   LIN {X 6.817, Y 34.224, Z 0.850} C_DIS
   LIN {X 6.879, Y 33.945, Z 0.850} C_DIS
   LIN {X 7.032, Y 33.271, Z 0.850} C_DIS
   LIN {X 7.088, Y 33.009, Z 0.850} C_DIS
   LIN {X 7.244, Y 32.286, Z 0.850} C_DIS
   LIN {X 7.311, Y 31.964, Z 0.850} C_DIS
   LIN {X 7.452, Y 31.279, Z 0.850} C_DIS
   LIN {X 7.589, Y 30.590, Z 0.850} C_DIS
   LIN {X 7.645, Y 30.301, Z 0.850} C_DIS
   LIN {X 7.699, Y 30.012, Z 0.850} C_DIS
   LIN {X 7.838, Y 29.273, Z 0.850} C_DIS
   LIN {X 7.890, Y 28.981, Z 0.850} C_DIS
   LIN {X 8.015, Y 28.279, Z 0.850} C_DIS
   LIN {X 8.061, Y 28.004, Z 0.850} C_DIS
   LIN {X 8.173, Y 27.343, Z 0.850} C_DIS
   LIN {X 8.220, Y 27.045, Z 0.850} C_DIS
   LIN {X 8.334, Y 26.335, Z 0.850} C_DIS
   LIN {X 8.379, Y 26.035, Z 0.850} C_DIS
   LIN {X 8.480, Y 25.364, Z 0.850} C_DIS
   LIN {X 8.523, Y 25.062, Z 0.850} C_DIS
   LIN {X 8.625, Y 24.342, Z 0.850} C_DIS
   LIN {X 8.662, Y 24.057, Z 0.850} C_DIS
   LIN {X 8.752, Y 23.378, Z 0.850} C_DIS
   LIN {X 8.790, Y 23.070, Z 0.850} C_DIS
   LIN {X 8.874, Y 22.388, Z 0.850} C_DIS
   LIN {X 8.912, Y 22.056, Z 0.850} C_DIS
   LIN {X 8.990, Y 21.369, Z 0.850} C_DIS
   LIN {X 9.021, Y 21.077, Z 0.850} C_DIS
   LIN {X 9.088, Y 20.433, Z 0.850} C_DIS
   LIN {X 9.119, Y 20.117, Z 0.850} C_DIS
   LIN {X 9.185, Y 19.423, Z 0.850} C_DIS
   LIN {X 9.213, Y 19.104, Z 0.850} C_DIS
   LIN {X 9.274, Y 18.407, Z 0.850} C_DIS
   LIN {X 9.297, Y 18.107, Z 0.850} C_DIS
   LIN {X 9.348, Y 17.453, Z 0.850} C_DIS
   LIN {X 9.370, Y 17.129, Z 0.850} C_DIS
   LIN {X 9.419, Y 16.426, Z 0.850} C_DIS
   LIN {X 9.438, Y 16.099, Z 0.850} C_DIS
   LIN {X 9.478, Y 15.439, Z 0.850} C_DIS
   LIN {X 9.494, Y 15.109, Z 0.850} C_DIS
   LIN {X 9.528, Y 14.447, Z 0.850} C_DIS
   LIN {X 9.541, Y 14.137, Z 0.850} C_DIS
   LIN {X 9.569, Y 13.472, Z 0.850} C_DIS
   LIN {X 9.580, Y 13.137, Z 0.850} C_DIS
   LIN {X 9.601, Y 12.470, Z 0.850} C_DIS
   LIN {X 9.610, Y 12.132, Z 0.850} C_DIS
   LIN {X 9.625, Y 11.463, Z 0.850} C_DIS
   LIN {X 9.630, Y 11.146, Z 0.850} C_DIS
   LIN {X 9.640, Y 10.474, Z 0.850} C_DIS
   LIN {X 9.642, Y 10.131, Z 0.850} C_DIS
   LIN {X 9.645, Y 9.504, Z 0.850} C_DIS
   LIN {X 9.645, Y 9.182, Z 0.850} C_DIS
   LIN {X 9.642, Y 8.509, Z 0.850} C_DIS
   LIN {X 9.638, Y 8.162, Z 0.850} C_DIS
   LIN {X 9.630, Y 7.539, Z 0.850} C_DIS
   LIN {X 9.623, Y 7.191, Z 0.850} C_DIS
   LIN {X 9.608, Y 6.491, Z 0.850} C_DIS
   LIN {X 9.598, Y 6.141, Z 0.850} C_DIS
   LIN {X 9.577, Y 5.502, Z 0.850} C_DIS
   LIN {X 9.565, Y 5.173, Z 0.850} C_DIS
   LIN {X 9.538, Y 4.519, Z 0.850} C_DIS
   LIN {X 9.522, Y 4.166, Z 0.850} C_DIS
   LIN {X 9.492, Y 3.556, Z 0.850} C_DIS
   LIN {X 9.472, Y 3.201, Z 0.850} C_DIS
   LIN {X 9.434, Y 2.546, Z 0.850} C_DIS
   LIN {X 9.411, Y 2.189, Z 0.850} C_DIS
   LIN {X 9.366, Y 1.536, Z 0.850} C_DIS
   LIN {X 9.340, Y 1.178, Z 0.850} C_DIS
   LIN {X 9.288, Y 0.517, Z 0.850} C_DIS
   LIN {X 9.261, Y 0.181, Z 0.850} C_DIS
   LIN {X 9.206, Y -0.450, Z 0.850} C_DIS
   LIN {X 9.173, Y -0.811, Z 0.850} C_DIS
   LIN {X 9.112, Y -1.448, Z 0.850} C_DIS
   LIN {X 9.075, Y -1.810, Z 0.850} C_DIS
   LIN {X 9.012, Y -2.415, Z 0.850} C_DIS
   LIN {X 8.972, Y -2.779, Z 0.850}
   LaserEnd_Ext()
   LIN {X 8.602, Y 12.437, Z 0.850}
   LaserStart_Ext()
   LIN {X 8.602, Y 6.300, Z 0.850}
   LaserEnd_Ext()
   LIN {X 7.602, Y -5.669, Z 0.850}
   LaserStart_Ext()
   LIN {X 7.602, Y 24.432, Z 0.850}
   LaserEnd_Ext()
   LIN {X 6.602, Y 30.425, Z 0.850}
   LaserStart_Ext()
   LIN {X 6.602, Y -11.632, Z 0.850}
   LaserEnd_Ext()
   LIN {X 5.602, Y -16.214, Z 0.850}
   LaserStart_Ext()
   LIN {X 5.602, Y 35.021, Z 0.850}
   LaserEnd_Ext()
   LIN {X 4.602, Y 38.415, Z 0.850}
   LaserStart_Ext()
   LIN {X 4.602, Y -20.060, Z 0.850}
   LaserEnd_Ext()
   LIN {X 3.602, Y -23.427, Z 0.850}
   LaserStart_Ext()
   LIN {X 3.602, Y 39.906, Z 0.850}
   LaserEnd_Ext()
   LIN {X 2.602, Y 40.540, Z 0.850}
   LaserStart_Ext()
   LIN {X 2.602, Y -25.992, Z 0.850}
   LaserEnd_Ext()
   LIN {X 1.602, Y -28.291, Z 0.850}
   LaserStart_Ext()
   LIN {X 1.602, Y 40.788, Z 0.850}
   LaserEnd_Ext()
   LIN {X 0.602, Y 40.704, Z 0.850}
   LaserStart_Ext()
   LIN {X 0.602, Y -29.565, Z 0.850}
   LaserEnd_Ext()
   LIN {X -0.398, Y -30.463, Z 0.850}
   LaserStart_Ext()
   LIN {X -0.398, Y 18.791, Z 0.850}
   LaserEnd_Ext()
   LIN {X -0.398, Y 23.726, Z 0.850}
   LaserStart_Ext()
   LIN {X -0.398, Y 40.289, Z 0.850}
   LaserEnd_Ext()
   LIN {X -1.398, Y 39.441, Z 0.850}
   LaserStart_Ext()
   LIN {X -1.398, Y 33.586, Z 0.850}
   LaserEnd_Ext()
   LIN {X -1.398, Y 8.945, Z 0.850}
   LaserStart_Ext()
   LIN {X -1.398, Y -31.122, Z 0.850}
   LaserEnd_Ext()
   LIN {X -2.398, Y -31.620, Z 0.850}
   LaserStart_Ext()
   LIN {X -2.398, Y 4.095, Z 0.850}
   LaserEnd_Ext()
   LIN {X -3.398, Y 0.392, Z 0.850}
   LaserStart_Ext()
   LIN {X -3.398, Y -32.036, Z 0.850}
   LaserEnd_Ext()
   LIN {X -4.398, Y -32.127, Z 0.850}
   LaserStart_Ext()
   LIN {X -4.398, Y -2.702, Z 0.850}
   LaserEnd_Ext()
   LIN {X -5.398, Y -5.406, Z 0.850}
   LaserStart_Ext()
   LIN {X -5.398, Y -32.235, Z 0.850}
   LaserEnd_Ext()
   LIN {X -6.398, Y -32.258, Z 0.850}
   LaserStart_Ext()
   LIN {X -6.398, Y -7.825, Z 0.850}
   LaserEnd_Ext()
   LIN {X -7.398, Y -10.028, Z 0.850}
   LaserStart_Ext()
   LIN {X -7.398, Y -32.049, Z 0.850}
   LaserEnd_Ext()
   LIN {X -8.398, Y -31.726, Z 0.850}
   LaserStart_Ext()
   LIN {X -8.398, Y -12.055, Z 0.850}
   LaserEnd_Ext()
   LIN {X -9.398, Y -13.938, Z 0.850}
   LaserStart_Ext()
   LIN {X -9.398, Y -31.348, Z 0.850}
   LaserEnd_Ext()
   LIN {X -10.398, Y -30.755, Z 0.850}
   LaserStart_Ext()
   LIN {X -10.398, Y -15.699, Z 0.850}
   LaserEnd_Ext()
   LIN {X -11.398, Y -17.353, Z 0.850}
   LaserStart_Ext()
   LIN {X -11.398, Y -29.935, Z 0.850}
   LaserEnd_Ext()
   LIN {X -12.398, Y -28.779, Z 0.850}
   LaserStart_Ext()
   LIN {X -12.398, Y -18.987, Z 0.850}
   LaserEnd_Ext()
   LIN {X -13.398, Y -20.925, Z 0.850}
   LaserStart_Ext()
   LIN {X -13.398, Y -26.767, Z 0.850}
   LaserEnd_Ext()
   LIN {X 3.579, Y 40.856, Z 1.700}
   LaserStart_Ext()
   LIN {X 4.137, Y 40.387, Z 1.700} C_DIS
   LIN {X 4.335, Y 40.229, Z 1.700} C_DIS
   LIN {X 4.824, Y 39.558, Z 1.700} C_DIS
   LIN {X 4.955, Y 39.387, Z 1.700} C_DIS
   LIN {X 5.275, Y 38.575, Z 1.700} C_DIS
   LIN {X 5.339, Y 38.424, Z 1.700} C_DIS
   LIN {X 5.362, Y 38.307, Z 1.700} C_DIS
   LIN {X 5.562, Y 37.562, Z 1.700} C_DIS
   LIN {X 5.589, Y 37.425, Z 1.700} C_DIS
   LIN {X 5.787, Y 36.662, Z 1.700} C_DIS
   LIN {X 5.838, Y 36.459, Z 1.700} C_DIS
   LIN {X 6.029, Y 35.692, Z 1.700} C_DIS
   LIN {X 6.081, Y 35.480, Z 1.700} C_DIS
   LIN {X 6.265, Y 34.710, Z 1.700} C_DIS
   LIN {X 6.317, Y 34.490, Z 1.700} C_DIS
   LIN {X 6.484, Y 33.761, Z 1.700} C_DIS
   LIN {X 6.532, Y 33.547, Z 1.700} C_DIS
   LIN {X 6.704, Y 32.769, Z 1.700} C_DIS
   LIN {X 6.754, Y 32.533, Z 1.700} C_DIS
   LIN {X 6.910, Y 31.798, Z 1.700} C_DIS
   LIN {X 6.957, Y 31.568, Z 1.700} C_DIS
   LIN {X 7.106, Y 30.830, Z 1.700} C_DIS
   LIN {X 7.152, Y 30.593, Z 1.700} C_DIS
   LIN {X 7.303, Y 29.805, Z 1.700} C_DIS
   LIN {X 7.352, Y 29.544, Z 1.700} C_DIS
   LIN {X 7.487, Y 28.800, Z 1.700} C_DIS
   LIN {X 7.532, Y 28.547, Z 1.700} C_DIS
   LIN {X 7.653, Y 27.847, Z 1.700} C_DIS
   LIN {X 7.694, Y 27.603, Z 1.700} C_DIS
   LIN {X 7.817, Y 26.854, Z 1.700} C_DIS
   LIN {X 7.859, Y 26.585, Z 1.700} C_DIS
   LIN {X 7.968, Y 25.881, Z 1.700} C_DIS
   LIN {X 8.007, Y 25.622, Z 1.700} C_DIS
   LIN {X 8.116, Y 24.869, Z 1.700} C_DIS
   LIN {X 8.156, Y 24.584, Z 1.700} C_DIS
   LIN {X 8.252, Y 23.877, Z 1.700} C_DIS
   LIN {X 8.288, Y 23.602, Z 1.700} C_DIS
   LIN {X 8.378, Y 22.893, Z 1.700} C_DIS
   LIN {X 8.412, Y 22.610, Z 1.700} C_DIS
   LIN {X 8.496, Y 21.901, Z 1.700} C_DIS
   LIN {X 8.528, Y 21.610, Z 1.700} C_DIS
   LIN {X 8.601, Y 20.947, Z 1.700} C_DIS
   LIN {X 8.629, Y 20.668, Z 1.700} C_DIS
   LIN {X 8.700, Y 19.957, Z 1.700} C_DIS
   LIN {X 8.729, Y 19.651, Z 1.700} C_DIS
   LIN {X 8.794, Y 18.938, Z 1.700} C_DIS
   LIN {X 8.820, Y 18.624, Z 1.700} C_DIS
   LIN {X 8.874, Y 17.959, Z 1.700} C_DIS
   LIN {X 8.897, Y 17.658, Z 1.700} C_DIS
   LIN {X 8.949, Y 16.945, Z 1.700} C_DIS
   LIN {X 8.971, Y 16.615, Z 1.700} C_DIS
   LIN {X 9.013, Y 15.949, Z 1.700} C_DIS
   LIN {X 9.031, Y 15.634, Z 1.700} C_DIS
   LIN {X 9.067, Y 14.968, Z 1.700} C_DIS
   LIN {X 9.082, Y 14.645, Z 1.700} C_DIS
   LIN {X 9.113, Y 13.980, Z 1.700} C_DIS
   LIN {X 9.125, Y 13.649, Z 1.700} C_DIS
   LIN {X 9.149, Y 12.984, Z 1.700} C_DIS
   LIN {X 9.160, Y 12.646, Z 1.700} C_DIS
   LIN {X 9.178, Y 11.981, Z 1.700} C_DIS
   LIN {X 9.185, Y 11.636, Z 1.700} C_DIS
   LIN {X 9.196, Y 10.972, Z 1.700} C_DIS
   LIN {X 9.201, Y 10.619, Z 1.700} C_DIS
   LIN {X 9.206, Y 10.002, Z 1.700} C_DIS
   LIN {X 9.207, Y 9.667, Z 1.700} C_DIS
   LIN {X 9.207, Y 9.004, Z 1.700} C_DIS
   LIN {X 9.204, Y 8.638, Z 1.700} C_DIS
   LIN {X 9.199, Y 8.023, Z 1.700} C_DIS
   LIN {X 9.193, Y 7.679, Z 1.700} C_DIS
   LIN {X 9.181, Y 7.018, Z 1.700} C_DIS
   LIN {X 9.171, Y 6.624, Z 1.700} C_DIS
   LIN {X 9.155, Y 6.011, Z 1.700} C_DIS
   LIN {X 9.142, Y 5.645, Z 1.700} C_DIS
   LIN {X 9.119, Y 5.016, Z 1.700} C_DIS
   LIN {X 9.103, Y 4.635, Z 1.700} C_DIS
   LIN {X 9.074, Y 4.021, Z 1.700} C_DIS
   LIN {X 9.056, Y 3.660, Z 1.700} C_DIS
   LIN {X 9.021, Y 3.042, Z 1.700} C_DIS
   LIN {X 8.997, Y 2.648, Z 1.700} C_DIS
   LIN {X 8.957, Y 2.026, Z 1.700} C_DIS
   LIN {X 8.929, Y 1.627, Z 1.700} C_DIS
   LIN {X 8.883, Y 1.001, Z 1.700} C_DIS
   LIN {X 8.850, Y 0.591, Z 1.700} C_DIS
   LIN {X 8.801, Y -0.004, Z 1.700} C_DIS
   LIN {X 8.765, Y -0.401, Z 1.700} C_DIS
   LIN {X 8.710, Y -0.999, Z 1.700} C_DIS
   LIN {X 8.670, Y -1.406, Z 1.700} C_DIS
   LIN {X 8.613, Y -1.971, Z 1.700} C_DIS
   LIN {X 8.571, Y -2.363, Z 1.700} C_DIS
   LIN {X 8.504, Y -2.966, Z 1.700} C_DIS
   LIN {X 8.454, Y -3.392, Z 1.700} C_DIS
   LIN {X 8.386, Y -3.962, Z 1.700} C_DIS
   LIN {X 8.334, Y -4.373, Z 1.700} C_DIS
   LIN {X 8.260, Y -4.945, Z 1.700} C_DIS
   LIN {X 8.204, Y -5.364, Z 1.700} C_DIS
   LIN {X 8.124, Y -5.938, Z 1.700} C_DIS
   LIN {X 8.063, Y -6.366, Z 1.700} C_DIS
   LIN {X 7.983, Y -6.905, Z 1.700} C_DIS
   LIN {X 7.920, Y -7.315, Z 1.700} C_DIS
   LIN {X 7.830, Y -7.891, Z 1.700} C_DIS
   LIN {X 7.757, Y -8.337, Z 1.700} C_DIS
   LIN {X 7.667, Y -8.879, Z 1.700} C_DIS
   LIN {X 7.594, Y -9.305, Z 1.700} C_DIS
   LIN {X 7.492, Y -9.884, Z 1.700} C_DIS
   LIN {X 7.408, Y -10.348, Z 1.700} C_DIS
   LIN {X 7.307, Y -10.892, Z 1.700} C_DIS
   LIN {X 7.222, Y -11.334, Z 1.700} C_DIS
   LIN {X 7.109, Y -11.915, Z 1.700} C_DIS
   LIN {X 7.012, Y -12.397, Z 1.700} C_DIS
   LIN {X 6.908, Y -12.905, Z 1.700} C_DIS
   LIN {X 6.818, Y -13.334, Z 1.700} C_DIS
   LIN {X 6.701, Y -13.879, Z 1.700} C_DIS
   LIN {X 6.599, Y -14.347, Z 1.700} C_DIS
   LIN {X 6.485, Y -14.856, Z 1.700} C_DIS
   LIN {X 6.383, Y -15.299, Z 1.700} C_DIS
   LIN {X 6.256, Y -15.845, Z 1.700} C_DIS
   LIN {X 6.140, Y -16.327, Z 1.700} C_DIS
   LIN {X 6.017, Y -16.837, Z 1.700} C_DIS
   LIN {X 5.903, Y -17.294, Z 1.700} C_DIS
   LIN {X 5.774, Y -17.804, Z 1.700} C_DIS
   LIN {X 5.654, Y -18.268, Z 1.700} C_DIS
   LIN {X 5.520, Y -18.777, Z 1.700} C_DIS
   LIN {X 5.394, Y -19.248, Z 1.700} C_DIS
   LIN {X 5.255, Y -19.757, Z 1.700} C_DIS
   LIN {X 5.122, Y -20.235, Z 1.700} C_DIS
   LIN {X 4.989, Y -20.707, Z 1.700} C_DIS
   LIN {X 4.859, Y -21.157, Z 1.700} C_DIS
   LIN {X 4.711, Y -21.665, Z 1.700} C_DIS
   LIN {X 4.565, Y -22.156, Z 1.700} C_DIS
   LIN {X 4.422, Y -22.627, Z 1.700} C_DIS
   LIN {X 4.280, Y -23.089, Z 1.700} C_DIS
   LIN {X 4.134, Y -23.560, Z 1.700} C_DIS
   LIN {X 3.985, Y -24.027, Z 1.700} C_DIS
   LIN {X 3.822, Y -24.533, Z 1.700} C_DIS
   LIN {X 3.655, Y -25.042, Z 1.700} C_DIS
   LIN {X 3.499, Y -25.512, Z 1.700} C_DIS
   LIN {X 3.296, Y -26.165, Z 1.700} C_DIS
   LIN {X 3.110, Y -26.708, Z 1.700} C_DIS
   LIN {X 2.898, Y -27.225, Z 1.700} C_DIS
   LIN {X 2.628, Y -27.815, Z 1.700} C_DIS
   LIN {X 2.354, Y -28.314, Z 1.700} C_DIS
   LIN {X 2.118, Y -28.700, Z 1.700} C_DIS
   LIN {X 1.790, Y -29.168, Z 1.700} C_DIS
   LIN {X 1.527, Y -29.505, Z 1.700} C_DIS
   LIN {X 1.139, Y -29.946, Z 1.700} C_DIS
   LIN {X 0.860, Y -30.235, Z 1.700} C_DIS
   LIN {X 0.425, Y -30.633, Z 1.700} C_DIS
   LIN {X 0.140, Y -30.871, Z 1.700} C_DIS
   LIN {X -0.367, Y -31.245, Z 1.700} C_DIS
   LIN {X -0.668, Y -31.445, Z 1.700} C_DIS
   LIN {X -1.235, Y -31.773, Z 1.700} C_DIS
   LIN {X -1.534, Y -31.928, Z 1.700} C_DIS
   LIN {X -2.141, Y -32.195, Z 1.700} C_DIS
   LIN {X -2.424, Y -32.304, Z 1.700} C_DIS
   LIN {X -3.090, Y -32.517, Z 1.700} C_DIS
   LIN {X -3.376, Y -32.593, Z 1.700} C_DIS
   LIN {X -4.071, Y -32.734, Z 1.700} C_DIS
   LIN {X -4.334, Y -32.775, Z 1.700} C_DIS
   LIN {X -5.050, Y -32.841, Z 1.700} C_DIS
   LIN {X -5.293, Y -32.852, Z 1.700} C_DIS
   LIN {X -6.043, Y -32.840, Z 1.700} C_DIS
   LIN {X -6.273, Y -32.825, Z 1.700} C_DIS
   LIN {X -7.047, Y -32.727, Z 1.700} C_DIS
   LIN {X -7.258, Y -32.690, Z 1.700} C_DIS
   LIN {X -8.021, Y -32.508, Z 1.700} C_DIS
   LIN {X -8.207, Y -32.453, Z 1.700} C_DIS
   LIN {X -8.971, Y -32.180, Z 1.700} C_DIS
   LIN {X -9.139, Y -32.110, Z 1.700} C_DIS
   LIN {X -9.871, Y -31.753, Z 1.700} C_DIS
   LIN {X -10.016, Y -31.673, Z 1.700} C_DIS
   LIN {X -10.717, Y -31.229, Z 1.700} C_DIS
   LIN {X -10.845, Y -31.139, Z 1.700} C_DIS
   LIN {X -11.509, Y -30.607, Z 1.700} C_DIS
   LIN {X -11.622, Y -30.506, Z 1.700} C_DIS
   LIN {X -12.222, Y -29.905, Z 1.700} C_DIS
   LIN {X -12.319, Y -29.797, Z 1.700} C_DIS
   LIN {X -12.864, Y -29.114, Z 1.700} C_DIS
   LIN {X -12.948, Y -28.996, Z 1.700} C_DIS
   LIN {X -13.394, Y -28.286, Z 1.700} C_DIS
   LIN {X -13.461, Y -28.164, Z 1.700} C_DIS
   LIN {X -13.834, Y -27.397, Z 1.700} C_DIS
   LIN {X -13.889, Y -27.264, Z 1.700} C_DIS
   LIN {X -14.171, Y -26.477, Z 1.700} C_DIS
   LIN {X -14.212, Y -26.336, Z 1.700} C_DIS
   LIN {X -14.411, Y -25.497, Z 1.700} C_DIS
   LIN {X -14.439, Y -25.341, Z 1.700} C_DIS
   LIN {X -14.539, Y -24.526, Z 1.700} C_DIS
   LIN {X -14.549, Y -24.360, Z 1.700} C_DIS
   LIN {X -14.560, Y -23.553, Z 1.700} C_DIS
   LIN {X -14.552, Y -23.375, Z 1.700} C_DIS
   LIN {X -14.473, Y -22.560, Z 1.700} C_DIS
   LIN {X -14.442, Y -22.363, Z 1.700} C_DIS
   LIN {X -14.284, Y -21.602, Z 1.700} C_DIS
   LIN {X -14.230, Y -21.403, Z 1.700} C_DIS
   LIN {X -13.996, Y -20.676, Z 1.700} C_DIS
   LIN {X -13.915, Y -20.471, Z 1.700} C_DIS
   LIN {X -13.602, Y -19.769, Z 1.700} C_DIS
   LIN {X -13.448, Y -19.474, Z 1.700} C_DIS
   LIN {X -13.060, Y -18.809, Z 1.700} C_DIS
   LIN {X -12.960, Y -18.666, Z 1.700} C_DIS
   LIN {X -12.567, Y -18.066, Z 1.700} C_DIS
   LIN {X -12.464, Y -17.914, Z 1.700} C_DIS
   LIN {X -12.058, Y -17.277, Z 1.700} C_DIS
   LIN {X -11.916, Y -17.050, Z 1.700} C_DIS
   LIN {X -11.526, Y -16.418, Z 1.700} C_DIS
   LIN {X -11.386, Y -16.188, Z 1.700} C_DIS
   LIN {X -11.022, Y -15.580, Z 1.700} C_DIS
   LIN {X -10.889, Y -15.354, Z 1.700} C_DIS
   LIN {X -10.512, Y -14.702, Z 1.700} C_DIS
   LIN {X -10.371, Y -14.455, Z 1.700} C_DIS
   LIN {X -10.015, Y -13.818, Z 1.700} C_DIS
   LIN {X -9.879, Y -13.572, Z 1.700} C_DIS
   LIN {X -9.533, Y -12.930, Z 1.700} C_DIS
   LIN {X -9.397, Y -12.676, Z 1.700} C_DIS
   LIN {X -9.061, Y -12.033, Z 1.700} C_DIS
   LIN {X -8.927, Y -11.773, Z 1.700} C_DIS
   LIN {X -8.605, Y -11.134, Z 1.700} C_DIS
   LIN {X -8.474, Y -10.871, Z 1.700} C_DIS
   LIN {X -8.166, Y -10.240, Z 1.700} C_DIS
   LIN {X -8.039, Y -9.975, Z 1.700} C_DIS
   LIN {X -7.747, Y -9.357, Z 1.700} C_DIS
   LIN {X -7.624, Y -9.093, Z 1.700} C_DIS
   LIN {X -7.332, Y -8.452, Z 1.700} C_DIS
   LIN {X -7.206, Y -8.173, Z 1.700} C_DIS
   LIN {X -6.932, Y -7.550, Z 1.700} C_DIS
   LIN {X -6.812, Y -7.273, Z 1.700} C_DIS
   LIN {X -6.540, Y -6.631, Z 1.700} C_DIS
   LIN {X -6.419, Y -6.340, Z 1.700} C_DIS
   LIN {X -6.150, Y -5.679, Z 1.700} C_DIS
   LIN {X -6.027, Y -5.374, Z 1.700} C_DIS
   LIN {X -5.778, Y -4.737, Z 1.700} C_DIS
   LIN {X -5.663, Y -4.437, Z 1.700} C_DIS
   LIN {X -5.435, Y -3.828, Z 1.700} C_DIS
   LIN {X -5.327, Y -3.537, Z 1.700} C_DIS
   LIN {X -5.103, Y -2.914, Z 1.700} C_DIS
   LIN {X -4.995, Y -2.610, Z 1.700} C_DIS
   LIN {X -4.776, Y -1.974, Z 1.700} C_DIS
   LIN {X -4.669, Y -1.658, Z 1.700} C_DIS
   LIN {X -4.456, Y -1.008, Z 1.700} C_DIS
   LIN {X -4.350, Y -0.679, Z 1.700} C_DIS
   LIN {X -4.157, Y -0.064, Z 1.700} C_DIS
   LIN {X -4.060, Y 0.254, Z 1.700} C_DIS
   LIN {X -3.873, Y 0.880, Z 1.700} C_DIS
   LIN {X -3.777, Y 1.208, Z 1.700} C_DIS
   LIN {X -3.597, Y 1.845, Z 1.700} C_DIS
   LIN {X -3.502, Y 2.186, Z 1.700} C_DIS
   LIN {X -3.329, Y 2.834, Z 1.700} C_DIS
   LIN {X -3.236, Y 3.188, Z 1.700} C_DIS
   LIN {X -3.083, Y 3.794, Z 1.700} C_DIS
   LIN {X -2.999, Y 4.131, Z 1.700} C_DIS
   LIN {X -2.841, Y 4.798, Z 1.700} C_DIS
   LIN {X -2.754, Y 5.174, Z 1.700} C_DIS
   LIN {X -2.615, Y 5.798, Z 1.700} C_DIS
   LIN {X -2.536, Y 6.162, Z 1.700} C_DIS
   LIN {X -2.415, Y 6.742, Z 1.700} C_DIS
   LIN {X -2.344, Y 7.092, Z 1.700} C_DIS
   LIN {X -2.220, Y 7.728, Z 1.700} C_DIS
   LIN {X -2.150, Y 8.099, Z 1.700} C_DIS
   LIN {X -2.038, Y 8.723, Z 1.700} C_DIS
   LIN {X -1.970, Y 9.111, Z 1.700} C_DIS
   LIN {X -1.868, Y 9.728, Z 1.700} C_DIS
   LIN {X -1.808, Y 10.105, Z 1.700} C_DIS
   LIN {X -1.717, Y 10.712, Z 1.700} C_DIS
   LIN {X -1.660, Y 11.100, Z 1.700} C_DIS
   LIN {X -1.579, Y 11.695, Z 1.700} C_DIS
   LIN {X -1.528, Y 12.083, Z 1.700} C_DIS
   LIN {X -1.456, Y 12.668, Z 1.700} C_DIS
   LIN {X -1.411, Y 13.053, Z 1.700} C_DIS
   LIN {X -1.344, Y 13.668, Z 1.700} C_DIS
   LIN {X -1.301, Y 14.080, Z 1.700} C_DIS
   LIN {X -1.244, Y 14.683, Z 1.700} C_DIS
   LIN {X -1.207, Y 15.095, Z 1.700} C_DIS
   LIN {X -1.159, Y 15.686, Z 1.700} C_DIS
   LIN {X -1.129, Y 16.097, Z 1.700} C_DIS
   LIN {X -1.090, Y 16.675, Z 1.700} C_DIS
   LIN {X -1.065, Y 17.085, Z 1.700} C_DIS
   LIN {X -1.034, Y 17.652, Z 1.700} C_DIS
   LIN {X -1.015, Y 18.060, Z 1.700} C_DIS
   LIN {X -0.992, Y 18.651, Z 1.700} C_DIS
   LIN {X -0.977, Y 19.084, Z 1.700} C_DIS
   LIN {X -0.962, Y 19.662, Z 1.700} C_DIS
   LIN {X -0.953, Y 20.093, Z 1.700} C_DIS
   LIN {X -0.947, Y 20.658, Z 1.700} C_DIS
   LIN {X -0.944, Y 21.086, Z 1.700} C_DIS
   LIN {X -0.945, Y 21.638, Z 1.700} C_DIS
   LIN {X -0.948, Y 22.062, Z 1.700} C_DIS
   LIN {X -0.957, Y 22.634, Z 1.700} C_DIS
   LIN {X -0.966, Y 23.082, Z 1.700} C_DIS
   LIN {X -0.982, Y 23.639, Z 1.700} C_DIS
   LIN {X -0.997, Y 24.083, Z 1.700} C_DIS
   LIN {X -1.022, Y 24.657, Z 1.700} C_DIS
   LIN {X -1.044, Y 25.122, Z 1.700} C_DIS
   LIN {X -1.074, Y 25.649, Z 1.700} C_DIS
   LIN {X -1.101, Y 26.084, Z 1.700} C_DIS
   LIN {X -1.139, Y 26.626, Z 1.700} C_DIS
   LIN {X -1.174, Y 27.081, Z 1.700} C_DIS
   LIN {X -1.221, Y 27.636, Z 1.700} C_DIS
   LIN {X -1.263, Y 28.110, Z 1.700} C_DIS
   LIN {X -1.316, Y 28.648, Z 1.700} C_DIS
   LIN {X -1.364, Y 29.114, Z 1.700} C_DIS
   LIN {X -1.423, Y 29.636, Z 1.700} C_DIS
   LIN {X -1.477, Y 30.095, Z 1.700} C_DIS
   LIN {X -1.544, Y 30.626, Z 1.700} C_DIS
   LIN {X -1.607, Y 31.101, Z 1.700} C_DIS
   LIN {X -1.679, Y 31.614, Z 1.700} C_DIS
   LIN {X -1.747, Y 32.080, Z 1.700} C_DIS
   LIN {X -1.827, Y 32.599, Z 1.700} C_DIS
   LIN {X -1.904, Y 33.078, Z 1.700} C_DIS
   LIN {X -1.992, Y 33.602, Z 1.700} C_DIS
   LIN {X -2.078, Y 34.093, Z 1.700} C_DIS
   LIN {X -2.170, Y 34.596, Z 1.700} C_DIS
   LIN {X -2.298, Y 35.163, Z 1.700} C_DIS
   LIN {X -2.412, Y 35.739, Z 1.700} C_DIS
   LIN {X -2.482, Y 36.308, Z 1.700} C_DIS
   LIN {X -2.536, Y 36.576, Z 1.700} C_DIS
   LIN {X -2.569, Y 36.778, Z 1.700} C_DIS
   LIN {X -2.647, Y 37.458, Z 1.700} C_DIS
   LIN {X -2.640, Y 37.788, Z 1.700} C_DIS
   LIN {X -2.575, Y 38.195, Z 1.700} C_DIS
   LIN {X -2.471, Y 38.624, Z 1.700} C_DIS
   LIN {X -2.259, Y 39.167, Z 1.700} C_DIS
   LIN {X -2.065, Y 39.532, Z 1.700} C_DIS
   LIN {X -1.608, Y 40.166, Z 1.700} C_DIS
   LIN {X -1.184, Y 40.614, Z 1.700} C_DIS
   LIN {X -0.712, Y 40.908, Z 1.700} C_DIS
   LIN {X -0.351, Y 41.138, Z 1.700} C_DIS
   LIN {X 0.222, Y 41.317, Z 1.700} C_DIS
   LIN {X 0.627, Y 41.451, Z 1.700} C_DIS
   LIN {X 1.268, Y 41.475, Z 1.700} C_DIS
   LIN {X 1.668, Y 41.499, Z 1.700} C_DIS
   LIN {X 2.337, Y 41.352, Z 1.700} C_DIS
   LIN {X 2.693, Y 41.284, Z 1.700} C_DIS
   LIN {X 3.308, Y 40.981, Z 1.700} C_DIS
   LIN {X 3.579, Y 40.856, Z 1.700}
   LaserEnd_Ext()
   LIN {X -0.839, Y 39.522, Z 1.700}
   LaserStart_Ext()
   LIN {X 3.614, Y 39.522, Z 1.700}
   LaserEnd_Ext()
   LIN {X 4.221, Y 38.522, Z 1.700}
   LaserStart_Ext()
   LIN {X -1.437, Y 38.522, Z 1.700}
   LaserEnd_Ext()
   LIN {X -1.646, Y 37.522, Z 1.700}
   LaserStart_Ext()
   LIN {X 4.537, Y 37.522, Z 1.700}
   LaserEnd_Ext()
   LIN {X 4.790, Y 36.522, Z 1.700}
   LaserStart_Ext()
   LIN {X -1.505, Y 36.522, Z 1.700}
   LaserEnd_Ext()
   LIN {X -1.350, Y 35.522, Z 1.700}
   LaserStart_Ext()
   LIN {X 5.041, Y 35.522, Z 1.700}
   LaserEnd_Ext()
   LIN {X 5.282, Y 34.522, Z 1.700}
   LaserStart_Ext()
   LIN {X -1.140, Y 34.522, Z 1.700}
   LaserEnd_Ext()
   LIN {X -0.964, Y 33.522, Z 1.700}
   LaserStart_Ext()
   LIN {X 5.513, Y 33.522, Z 1.700}
   LaserEnd_Ext()
   LIN {X 5.734, Y 32.522, Z 1.700}
   LaserStart_Ext()
   LIN {X -0.803, Y 32.522, Z 1.700}
   LaserEnd_Ext()
   LIN {X -0.656, Y 31.522, Z 1.700}
   LaserStart_Ext()
   LIN {X 5.945, Y 31.522, Z 1.700}
   LaserEnd_Ext()
   LIN {X 6.147, Y 30.522, Z 1.700}
   LaserStart_Ext()
   LIN {X -0.523, Y 30.522, Z 1.700}
   LaserEnd_Ext()
   LIN {X -0.404, Y 29.522, Z 1.700}
   LaserStart_Ext()
   LIN {X 6.339, Y 29.522, Z 1.700}
   LaserEnd_Ext()
   LIN {X 6.521, Y 28.522, Z 1.700}
   LaserStart_Ext()
   LIN {X -0.299, Y 28.522, Z 1.700}
   LaserEnd_Ext()
   LIN {X -0.207, Y 27.522, Z 1.700}
   LaserStart_Ext()
   LIN {X 6.694, Y 27.522, Z 1.700}
   LaserEnd_Ext()
   LIN {X 6.857, Y 26.522, Z 1.700}
   LaserStart_Ext()
   LIN {X -0.130, Y 26.522, Z 1.700}
   LaserEnd_Ext()
   LIN {X -0.066, Y 25.522, Z 1.700}
   LaserStart_Ext()
   LIN {X 7.011, Y 25.522, Z 1.700}
   LaserEnd_Ext()
   LIN {X 7.155, Y 24.522, Z 1.700}
   LaserStart_Ext()
   LIN {X -0.015, Y 24.522, Z 1.700}
   LaserEnd_Ext()
   LIN {X 0.022, Y 23.522, Z 1.700}
   LaserStart_Ext()
   LIN {X 7.290, Y 23.522, Z 1.700}
   LaserEnd_Ext()
   LIN {X 7.416, Y 22.522, Z 1.700}
   LaserStart_Ext()
   LIN {X 0.045, Y 22.522, Z 1.700}
   LaserEnd_Ext()
   LIN {X 0.055, Y 21.522, Z 1.700}
   LaserStart_Ext()
   LIN {X 7.532, Y 21.522, Z 1.700}
   LaserEnd_Ext()
   LIN {X 7.639, Y 20.522, Z 1.700}
   LaserStart_Ext()
   LIN {X 0.052, Y 20.522, Z 1.700}
   LaserEnd_Ext()
   LIN {X 0.035, Y 19.522, Z 1.700}
   LaserStart_Ext()
   LIN {X 7.737, Y 19.522, Z 1.700}
   LaserEnd_Ext()
   LIN {X 7.825, Y 18.522, Z 1.700}
   LaserStart_Ext()
   LIN {X 0.004, Y 18.522, Z 1.700}
   LaserEnd_Ext()
   LIN {X -0.040, Y 17.522, Z 1.700}
   LaserStart_Ext()
   LIN {X 7.904, Y 17.522, Z 1.700}
   LaserEnd_Ext()
   LIN {X 7.975, Y 16.522, Z 1.700}
   LaserStart_Ext()
   LIN {X -0.098, Y 16.522, Z 1.700}
   LaserEnd_Ext()
   LIN {X -0.169, Y 15.522, Z 1.700}
   LaserStart_Ext()
   LIN {X 8.035, Y 15.522, Z 1.700}
   LaserEnd_Ext()
   LIN {X 8.087, Y 14.522, Z 1.700}
   LaserStart_Ext()
   LIN {X -0.255, Y 14.522, Z 1.700}
   LaserEnd_Ext()
   LIN {X -0.354, Y 13.522, Z 1.700}
   LaserStart_Ext()
   LIN {X 8.129, Y 13.522, Z 1.700}
   LaserEnd_Ext()
   LIN {X 8.163, Y 12.522, Z 1.700}
   LaserStart_Ext()
   LIN {X -0.466, Y 12.522, Z 1.700}
   LaserEnd_Ext()
   LIN {X -0.593, Y 11.522, Z 1.700}
   LaserStart_Ext()
   LIN {X 8.187, Y 11.522, Z 1.700}
   LaserEnd_Ext()
   LIN {X 8.201, Y 10.522, Z 1.700}
   LaserStart_Ext()
   LIN {X -0.734, Y 10.522, Z 1.700}
   LaserEnd_Ext()
   LIN {X -0.889, Y 9.522, Z 1.700}
   LaserStart_Ext()
   LIN {X 8.207, Y 9.522, Z 1.700}
   LaserEnd_Ext()
   LIN {X 8.203, Y 8.522, Z 1.700}
   LaserStart_Ext()
   LIN {X -1.058, Y 8.522, Z 1.700}
   LaserEnd_Ext()
   LIN {X -1.242, Y 7.522, Z 1.700}
   LaserStart_Ext()
   LIN {X 8.190, Y 7.522, Z 1.700}
   LaserEnd_Ext()
   LIN {X 8.168, Y 6.522, Z 1.700}
   LaserStart_Ext()
   LIN {X -1.439, Y 6.522, Z 1.700}
   LaserEnd_Ext()
   LIN {X -1.652, Y 5.522, Z 1.700}
   LaserStart_Ext()
   LIN {X 8.137, Y 5.522, Z 1.700}
   LaserEnd_Ext()
   LIN {X 8.096, Y 4.522, Z 1.700}
   LaserStart_Ext()
   LIN {X -1.879, Y 4.522, Z 1.700}
   LaserEnd_Ext()
   LIN {X -2.121, Y 3.522, Z 1.700}
   LaserStart_Ext()
   LIN {X 8.046, Y 3.522, Z 1.700}
   LaserEnd_Ext()
   LIN {X 7.987, Y 2.522, Z 1.700}
   LaserStart_Ext()
   LIN {X -2.377, Y 2.522, Z 1.700}
   LaserEnd_Ext()
   LIN {X -2.649, Y 1.522, Z 1.700}
   LaserStart_Ext()
   LIN {X 7.919, Y 1.522, Z 1.700}
   LaserEnd_Ext()
   LIN {X 7.841, Y 0.522, Z 1.700}
   LaserStart_Ext()
   LIN {X -2.936, Y 0.522, Z 1.700}
   LaserEnd_Ext()
   LIN {X -3.239, Y -0.478, Z 1.700}
   LaserStart_Ext()
   LIN {X 7.754, Y -0.478, Z 1.700}
   LaserEnd_Ext()
   LIN {X 7.658, Y -1.478, Z 1.700}
   LaserStart_Ext()
   LIN {X -3.558, Y -1.478, Z 1.700}
   LaserEnd_Ext()
   LIN {X -3.892, Y -2.478, Z 1.700}
   LaserStart_Ext()
   LIN {X 7.552, Y -2.478, Z 1.700}
   LaserEnd_Ext()
   LIN {X 7.437, Y -3.478, Z 1.700}
   LaserStart_Ext()
   LIN {X -4.243, Y -3.478, Z 1.700}
   LaserEnd_Ext()
   LIN {X -4.610, Y -4.478, Z 1.700}
   LaserStart_Ext()
   LIN {X 7.312, Y -4.478, Z 1.700}
   LaserEnd_Ext()
   LIN {X 7.178, Y -5.478, Z 1.700}
   LaserStart_Ext()
   LIN {X -4.994, Y -5.478, Z 1.700}
   LaserEnd_Ext()
   LIN {X -5.395, Y -6.478, Z 1.700}
   LaserStart_Ext()
   LIN {X 7.035, Y -6.478, Z 1.700}
   LaserEnd_Ext()
   LIN {X 6.882, Y -7.478, Z 1.700}
   LaserStart_Ext()
   LIN {X -5.813, Y -7.478, Z 1.700}
   LaserEnd_Ext()
   LIN {X -6.248, Y -8.478, Z 1.700}
   LaserStart_Ext()
   LIN {X 6.720, Y -8.478, Z 1.700}
   LaserEnd_Ext()
   LIN {X 6.548, Y -9.478, Z 1.700}
   LaserStart_Ext()
   LIN {X -6.701, Y -9.478, Z 1.700}
   LaserEnd_Ext()
   LIN {X -7.171, Y -10.478, Z 1.700}
   LaserStart_Ext()
   LIN {X 6.367, Y -10.478, Z 1.700}
   LaserEnd_Ext()
   LIN {X 6.176, Y -11.478, Z 1.700}
   LaserStart_Ext()
   LIN {X -7.659, Y -11.478, Z 1.700}
   LaserEnd_Ext()
   LIN {X -8.166, Y -12.478, Z 1.700}
   LaserStart_Ext()
   LIN {X 5.975, Y -12.478, Z 1.700}
   LaserEnd_Ext()
   LIN {X 5.765, Y -13.478, Z 1.700}
   LaserStart_Ext()
   LIN {X -8.692, Y -13.478, Z 1.700}
   LaserEnd_Ext()
   LIN {X -9.239, Y -14.478, Z 1.700}
   LaserStart_Ext()
   LIN {X 5.545, Y -14.478, Z 1.700}
   LaserEnd_Ext()
   LIN {X 5.315, Y -15.478, Z 1.700}
   LaserStart_Ext()
   LIN {X -9.806, Y -15.478, Z 1.700}
   LaserEnd_Ext()
   LIN {X -10.394, Y -16.478, Z 1.700}
   LaserStart_Ext()
   LIN {X 5.075, Y -16.478, Z 1.700}
   LaserEnd_Ext()
   LIN {X 4.825, Y -17.478, Z 1.700}
   LaserStart_Ext()
   LIN {X -11.005, Y -17.478, Z 1.700}
   LaserEnd_Ext()
   LIN {X -11.639, Y -18.478, Z 1.700}
   LaserStart_Ext()
   LIN {X 4.565, Y -18.478, Z 1.700}
   LaserEnd_Ext()
   LIN {X 4.295, Y -19.478, Z 1.700}
   LaserStart_Ext()
   LIN {X -12.292, Y -19.478, Z 1.700}
   LaserEnd_Ext()
   LIN {X -12.823, Y -20.478, Z 1.700}
   LaserStart_Ext()
   LIN {X 4.014, Y -20.478, Z 1.700}
   LaserEnd_Ext()
   LIN {X 3.723, Y -21.478, Z 1.700}
   LaserStart_Ext()
   LIN {X -13.203, Y -21.478, Z 1.700}
   LaserEnd_Ext()
   LIN {X -13.445, Y -22.478, Z 1.700}
   LaserStart_Ext()
   LIN {X 3.422, Y -22.478, Z 1.700}
   LaserEnd_Ext()
   LIN {X 3.110, Y -23.478, Z 1.700}
   LaserStart_Ext()
   LIN {X -13.556, Y -23.478, Z 1.700}
   LaserEnd_Ext()
   LIN {X -13.538, Y -24.478, Z 1.700}
   LaserStart_Ext()
   LIN {X 2.788, Y -24.478, Z 1.700}
   LaserEnd_Ext()
   LIN {X 2.462, Y -25.478, Z 1.700}
   LaserStart_Ext()
   LIN {X -13.388, Y -25.478, Z 1.700}
   LaserEnd_Ext()
   LIN {X -13.108, Y -26.478, Z 1.700}
   LaserStart_Ext()
   LIN {X 2.123, Y -26.478, Z 1.700}
   LaserEnd_Ext()
   LIN {X 1.672, Y -27.478, Z 1.700}
   LaserStart_Ext()
   LIN {X -12.682, Y -27.478, Z 1.700}
   LaserEnd_Ext()
   LIN {X -12.089, Y -28.478, Z 1.700}
   LaserStart_Ext()
   LIN {X 1.052, Y -28.478, Z 1.700}
   LaserEnd_Ext()
   LIN {X 0.200, Y -29.478, Z 1.700}
   LaserStart_Ext()
   LIN {X -11.235, Y -29.478, Z 1.700}
   LaserEnd_Ext()
   LIN {X -10.034, Y -30.478, Z 1.700}
   LaserStart_Ext()
   LIN {X -1.020, Y -30.478, Z 1.700}
   LaserEnd_Ext()
   LIN {X -3.125, Y -31.478, Z 1.700}
   LaserStart_Ext()
   LIN {X -7.964, Y -31.478, Z 1.700}
   LaserEnd_Ext()
   LIN {X 8.361, Y 22.380, Z 2.550}
   LaserStart_Ext()
   LIN {X 8.392, Y 22.114, Z 2.550} C_DIS
   LIN {X 8.473, Y 21.404, Z 2.550} C_DIS
   LIN {X 8.501, Y 21.149, Z 2.550} C_DIS
   LIN {X 8.575, Y 20.444, Z 2.550} C_DIS
   LIN {X 8.603, Y 20.163, Z 2.550} C_DIS
   LIN {X 8.674, Y 19.429, Z 2.550} C_DIS
   LIN {X 8.700, Y 19.140, Z 2.550} C_DIS
   LIN {X 8.761, Y 18.431, Z 2.550} C_DIS
   LIN {X 8.784, Y 18.154, Z 2.550} C_DIS
   LIN {X 8.839, Y 17.444, Z 2.550} C_DIS
   LIN {X 8.861, Y 17.139, Z 2.550} C_DIS
   LIN {X 8.910, Y 16.428, Z 2.550} C_DIS
   LIN {X 8.928, Y 16.137, Z 2.550} C_DIS
   LIN {X 8.969, Y 15.451, Z 2.550} C_DIS
   LIN {X 8.985, Y 15.151, Z 2.550} C_DIS
   LIN {X 9.020, Y 14.465, Z 2.550} C_DIS
   LIN {X 9.033, Y 14.159, Z 2.550} C_DIS
   LIN {X 9.062, Y 13.473, Z 2.550} C_DIS
   LIN {X 9.073, Y 13.159, Z 2.550} C_DIS
   LIN {X 9.095, Y 12.476, Z 2.550} C_DIS
   LIN {X 9.104, Y 12.149, Z 2.550} C_DIS
   LIN {X 9.120, Y 11.467, Z 2.550} C_DIS
   LIN {X 9.125, Y 11.138, Z 2.550} C_DIS
   LIN {X 9.135, Y 10.477, Z 2.550} C_DIS
   LIN {X 9.137, Y 10.164, Z 2.550} C_DIS
   LIN {X 9.141, Y 9.505, Z 2.550} C_DIS
   LIN {X 9.141, Y 9.161, Z 2.550} C_DIS
   LIN {X 9.138, Y 8.507, Z 2.550} C_DIS
   LIN {X 9.135, Y 8.181, Z 2.550} C_DIS
   LIN {X 9.126, Y 7.520, Z 2.550} C_DIS
   LIN {X 9.119, Y 7.153, Z 2.550} C_DIS
   LIN {X 9.105, Y 6.491, Z 2.550} C_DIS
   LIN {X 9.095, Y 6.143, Z 2.550} C_DIS
   LIN {X 9.075, Y 5.506, Z 2.550} C_DIS
   LIN {X 9.061, Y 5.141, Z 2.550} C_DIS
   LIN {X 9.036, Y 4.518, Z 2.550} C_DIS
   LIN {X 9.019, Y 4.161, Z 2.550} C_DIS
   LIN {X 8.988, Y 3.537, Z 2.550} C_DIS
   LIN {X 8.968, Y 3.169, Z 2.550} C_DIS
   LIN {X 8.930, Y 2.527, Z 2.550} C_DIS
   LIN {X 8.905, Y 2.148, Z 2.550} C_DIS
   LIN {X 8.862, Y 1.506, Z 2.550} C_DIS
   LIN {X 8.832, Y 1.117, Z 2.550} C_DIS
   LIN {X 8.784, Y 0.489, Z 2.550} C_DIS
   LIN {X 8.752, Y 0.111, Z 2.550} C_DIS
   LIN {X 8.699, Y -0.502, Z 2.550} C_DIS
   LIN {X 8.663, Y -0.890, Z 2.550} C_DIS
   LIN {X 8.605, Y -1.488, Z 2.550} C_DIS
   LIN {X 8.567, Y -1.862, Z 2.550} C_DIS
   LIN {X 8.504, Y -2.462, Z 2.550} C_DIS
   LIN {X 8.459, Y -2.869, Z 2.550} C_DIS
   LIN {X 8.390, Y -3.472, Z 2.550} C_DIS
   LIN {X 8.343, Y -3.865, Z 2.550} C_DIS
   LIN {X 8.270, Y -4.451, Z 2.550} C_DIS
   LIN {X 8.218, Y -4.853, Z 2.550} C_DIS
   LIN {X 8.140, Y -5.440, Z 2.550} C_DIS
   LIN {X 8.083, Y -5.853, Z 2.550} C_DIS
   LIN {X 8.002, Y -6.423, Z 2.550} C_DIS
   LIN {X 7.943, Y -6.816, Z 2.550} C_DIS
   LIN {X 7.857, Y -7.389, Z 2.550} C_DIS
   LIN {X 7.789, Y -7.818, Z 2.550} C_DIS
   LIN {X 7.697, Y -8.391, Z 2.550} C_DIS
   LIN {X 7.629, Y -8.802, Z 2.550} C_DIS
   LIN {X 7.531, Y -9.376, Z 2.550} C_DIS
   LIN {X 7.452, Y -9.823, Z 2.550} C_DIS
   LIN {X 7.349, Y -10.398, Z 2.550} C_DIS
   LIN {X 7.270, Y -10.826, Z 2.550} C_DIS
   LIN {X 7.173, Y -11.342, Z 2.550} C_DIS
   LIN {X 7.058, Y -11.927, Z 2.550} C_DIS
   LIN {X 6.959, Y -12.424, Z 2.550} C_DIS
   LIN {X 6.874, Y -12.840, Z 2.550} C_DIS
   LIN {X 6.761, Y -13.379, Z 2.550} C_DIS
   LIN {X 6.664, Y -13.832, Z 2.550} C_DIS
   LIN {X 6.547, Y -14.371, Z 2.550} C_DIS
   LIN {X 6.450, Y -14.802, Z 2.550} C_DIS
   LIN {X 6.328, Y -15.340, Z 2.550} C_DIS
   LIN {X 6.218, Y -15.810, Z 2.550} C_DIS
   LIN {X 6.090, Y -16.348, Z 2.550} C_DIS
   LIN {X 5.981, Y -16.794, Z 2.550} C_DIS
   LIN {X 5.853, Y -17.313, Z 2.550} C_DIS
   LIN {X 5.738, Y -17.766, Z 2.550} C_DIS
   LIN {X 5.605, Y -18.287, Z 2.550} C_DIS
   LIN {X 5.484, Y -18.748, Z 2.550} C_DIS
   LIN {X 5.346, Y -19.263, Z 2.550} C_DIS
   LIN {X 5.219, Y -19.731, Z 2.550} C_DIS
   LIN {X 5.081, Y -20.229, Z 2.550} C_DIS
   LIN {X 4.956, Y -20.670, Z 2.550} C_DIS
   LIN {X 4.814, Y -21.168, Z 2.550} C_DIS
   LIN {X 4.673, Y -21.650, Z 2.550} C_DIS
   LIN {X 4.525, Y -22.149, Z 2.550} C_DIS
   LIN {X 4.388, Y -22.602, Z 2.550} C_DIS
   LIN {X 4.243, Y -23.078, Z 2.550} C_DIS
   LIN {X 4.099, Y -23.537, Z 2.550} C_DIS
   LIN {X 3.970, Y -23.949, Z 2.550} C_DIS
   LIN {X 3.752, Y -24.624, Z 2.550} C_DIS
   LIN {X 3.628, Y -25.006, Z 2.550} C_DIS
   LIN {X 3.398, Y -25.697, Z 2.550} C_DIS
   LIN {X 3.274, Y -26.066, Z 2.550} C_DIS
   LIN {X 3.074, Y -26.649, Z 2.550} C_DIS
   LIN {X 2.931, Y -26.999, Z 2.550} C_DIS
   LIN {X 2.711, Y -27.541, Z 2.550} C_DIS
   LIN {X 2.425, Y -28.070, Z 2.550} C_DIS
   LIN {X 2.040, Y -28.720, Z 2.550} C_DIS
   LIN {X 1.783, Y -29.089, Z 2.550} C_DIS
   LIN {X 1.434, Y -29.526, Z 2.550} C_DIS
   LIN {X 1.155, Y -29.847, Z 2.550} C_DIS
   LIN {X 0.751, Y -30.254, Z 2.550} C_DIS
   LIN {X 0.465, Y -30.519, Z 2.550} C_DIS
   LIN {X 0.001, Y -30.896, Z 2.550} C_DIS
   LIN {X -0.301, Y -31.122, Z 2.550} C_DIS
   LIN {X -0.833, Y -31.465, Z 2.550} C_DIS
   LIN {X -1.136, Y -31.643, Z 2.550} C_DIS
   LIN {X -1.716, Y -31.932, Z 2.550} C_DIS
   LIN {X -2.005, Y -32.062, Z 2.550} C_DIS
   LIN {X -2.637, Y -32.297, Z 2.550} C_DIS
   LIN {X -2.922, Y -32.389, Z 2.550} C_DIS
   LIN {X -3.603, Y -32.562, Z 2.550} C_DIS
   LIN {X -3.870, Y -32.618, Z 2.550} C_DIS
   LIN {X -4.573, Y -32.718, Z 2.550} C_DIS
   LIN {X -4.821, Y -32.742, Z 2.550} C_DIS
   LIN {X -5.551, Y -32.766, Z 2.550} C_DIS
   LIN {X -5.783, Y -32.763, Z 2.550} C_DIS
   LIN {X -6.543, Y -32.706, Z 2.550} C_DIS
   LIN {X -6.757, Y -32.680, Z 2.550} C_DIS
   LIN {X -7.524, Y -32.537, Z 2.550} C_DIS
   LIN {X -7.713, Y -32.492, Z 2.550} C_DIS
   LIN {X -8.474, Y -32.263, Z 2.550} C_DIS
   LIN {X -8.644, Y -32.203, Z 2.550} C_DIS
   LIN {X -9.389, Y -31.886, Z 2.550} C_DIS
   LIN {X -9.537, Y -31.815, Z 2.550} C_DIS
   LIN {X -10.245, Y -31.416, Z 2.550} C_DIS
   LIN {X -10.383, Y -31.330, Z 2.550} C_DIS
   LIN {X -11.055, Y -30.848, Z 2.550} C_DIS
   LIN {X -11.178, Y -30.750, Z 2.550} C_DIS
   LIN {X -11.801, Y -30.191, Z 2.550} C_DIS
   LIN {X -11.902, Y -30.090, Z 2.550} C_DIS
   LIN {X -12.465, Y -29.460, Z 2.550} C_DIS
   LIN {X -12.558, Y -29.343, Z 2.550} C_DIS
   LIN {X -13.048, Y -28.654, Z 2.550} C_DIS
   LIN {X -13.122, Y -28.536, Z 2.550} C_DIS
   LIN {X -13.527, Y -27.807, Z 2.550} C_DIS
   LIN {X -13.588, Y -27.683, Z 2.550} C_DIS
   LIN {X -13.914, Y -26.906, Z 2.550} C_DIS
   LIN {X -13.960, Y -26.779, Z 2.550} C_DIS
   LIN {X -14.201, Y -25.970, Z 2.550} C_DIS
   LIN {X -14.235, Y -25.828, Z 2.550} C_DIS
   LIN {X -14.384, Y -25.009, Z 2.550} C_DIS
   LIN {X -14.402, Y -24.859, Z 2.550} C_DIS
   LIN {X -14.460, Y -24.050, Z 2.550} C_DIS
   LIN {X -14.462, Y -23.887, Z 2.550} C_DIS
   LIN {X -14.431, Y -23.077, Z 2.550} C_DIS
   LIN {X -14.413, Y -22.895, Z 2.550} C_DIS
   LIN {X -14.299, Y -22.113, Z 2.550} C_DIS
   LIN {X -14.260, Y -21.926, Z 2.550} C_DIS
   LIN {X -14.067, Y -21.178, Z 2.550} C_DIS
   LIN {X -14.003, Y -20.983, Z 2.550} C_DIS
   LIN {X -13.640, Y -20.086, Z 2.550} C_DIS
   LIN {X -13.452, Y -19.669, Z 2.550} C_DIS
   LIN {X -13.219, Y -19.272, Z 2.550} C_DIS
   LIN {X -12.958, Y -18.826, Z 2.550} C_DIS
   LIN {X -12.709, Y -18.447, Z 2.550} C_DIS
   LIN {X -12.352, Y -17.896, Z 2.550} C_DIS
   LIN {X -11.977, Y -17.310, Z 2.550} C_DIS
   LIN {X -11.724, Y -16.897, Z 2.550} C_DIS
   LIN {X -11.577, Y -16.660, Z 2.550} C_DIS
   LIN {X -11.207, Y -16.049, Z 2.550} C_DIS
   LIN {X -11.067, Y -15.815, Z 2.550} C_DIS
   LIN {X -10.703, Y -15.195, Z 2.550} C_DIS
   LIN {X -10.554, Y -14.938, Z 2.550} C_DIS
   LIN {X -10.194, Y -14.305, Z 2.550} C_DIS
   LIN {X -10.051, Y -14.049, Z 2.550} C_DIS
   LIN {X -9.706, Y -13.421, Z 2.550} C_DIS
   LIN {X -9.563, Y -13.157, Z 2.550} C_DIS
   LIN {X -9.228, Y -12.527, Z 2.550} C_DIS
   LIN {X -9.087, Y -12.257, Z 2.550} C_DIS
   LIN {X -8.764, Y -11.628, Z 2.550} C_DIS
   LIN {X -8.626, Y -11.354, Z 2.550} C_DIS
   LIN {X -8.317, Y -10.732, Z 2.550} C_DIS
   LIN {X -8.182, Y -10.455, Z 2.550} C_DIS
   LIN {X -7.889, Y -9.844, Z 2.550} C_DIS
   LIN {X -7.758, Y -9.567, Z 2.550} C_DIS
   LIN {X -7.473, Y -8.952, Z 2.550} C_DIS
   LIN {X -7.339, Y -8.659, Z 2.550} C_DIS
   LIN {X -7.064, Y -8.042, Z 2.550} C_DIS
   LIN {X -6.936, Y -7.752, Z 2.550} C_DIS
   LIN {X -6.670, Y -7.134, Z 2.550} C_DIS
   LIN {X -6.541, Y -6.829, Z 2.550} C_DIS
   LIN {X -6.278, Y -6.193, Z 2.550} C_DIS
   LIN {X -6.147, Y -5.873, Z 2.550} C_DIS
   LIN {X -5.895, Y -5.240, Z 2.550} C_DIS
   LIN {X -5.772, Y -4.925, Z 2.550} C_DIS
   LIN {X -5.541, Y -4.318, Z 2.550} C_DIS
   LIN {X -5.425, Y -4.012, Z 2.550} C_DIS
   LIN {X -5.206, Y -3.412, Z 2.550} C_DIS
   LIN {X -5.091, Y -3.093, Z 2.550} C_DIS
   LIN {X -4.876, Y -2.481, Z 2.550} C_DIS
   LIN {X -4.761, Y -2.148, Z 2.550} C_DIS
   LIN {X -4.552, Y -1.523, Z 2.550} C_DIS
   LIN {X -4.438, Y -1.177, Z 2.550} C_DIS
   LIN {X -4.241, Y -0.563, Z 2.550} C_DIS
   LIN {X -4.136, Y -0.229, Z 2.550} C_DIS
   LIN {X -3.953, Y 0.373, Z 2.550} C_DIS
   LIN {X -3.849, Y 0.719, Z 2.550} C_DIS
   LIN {X -3.689, Y 1.269, Z 2.550} C_DIS
   LIN {X -3.552, Y 1.751, Z 2.550} C_DIS
   LIN {X -3.399, Y 2.312, Z 2.550} C_DIS
   LIN {X -3.299, Y 2.685, Z 2.550} C_DIS
   LIN {X -3.142, Y 3.292, Z 2.550} C_DIS
   LIN {X -3.051, Y 3.648, Z 2.550} C_DIS
   LIN {X -2.901, Y 4.260, Z 2.550} C_DIS
   LIN {X -2.806, Y 4.659, Z 2.550} C_DIS
   LIN {X -2.663, Y 5.283, Z 2.550} C_DIS
   LIN {X -2.578, Y 5.664, Z 2.550} C_DIS
   LIN {X -2.451, Y 6.254, Z 2.550} C_DIS
   LIN {X -2.375, Y 6.615, Z 2.550} C_DIS
   LIN {X -2.258, Y 7.199, Z 2.550} C_DIS
   LIN {X -2.179, Y 7.603, Z 2.550} C_DIS
   LIN {X -2.067, Y 8.205, Z 2.550} C_DIS
   LIN {X -1.994, Y 8.609, Z 2.550} C_DIS
   LIN {X -1.892, Y 9.203, Z 2.550} C_DIS
   LIN {X -1.824, Y 9.612, Z 2.550} C_DIS
   LIN {X -1.733, Y 10.193, Z 2.550} C_DIS
   LIN {X -1.671, Y 10.603, Z 2.550} C_DIS
   LIN {X -1.588, Y 11.180, Z 2.550} C_DIS
   LIN {X -1.532, Y 11.591, Z 2.550} C_DIS
   LIN {X -1.459, Y 12.155, Z 2.550} C_DIS
   LIN {X -1.408, Y 12.566, Z 2.550} C_DIS
   LIN {X -1.343, Y 13.137, Z 2.550} C_DIS
   LIN {X -1.294, Y 13.578, Z 2.550} C_DIS
   LIN {X -1.236, Y 14.158, Z 2.550} C_DIS
   LIN {X -1.194, Y 14.598, Z 2.550} C_DIS
   LIN {X -1.145, Y 15.165, Z 2.550} C_DIS
   LIN {X -1.109, Y 15.605, Z 2.550} C_DIS
   LIN {X -1.068, Y 16.159, Z 2.550} C_DIS
   LIN {X -1.039, Y 16.598, Z 2.550} C_DIS
   LIN {X -1.007, Y 17.140, Z 2.550} C_DIS
   LIN {X -0.983, Y 17.578, Z 2.550} C_DIS
   LIN {X -0.958, Y 18.125, Z 2.550} C_DIS
   LIN {X -0.939, Y 18.591, Z 2.550} C_DIS
   LIN {X -0.922, Y 19.142, Z 2.550} C_DIS
   LIN {X -0.910, Y 19.605, Z 2.550} C_DIS
   LIN {X -0.900, Y 20.143, Z 2.550} C_DIS
   LIN {X -0.894, Y 20.603, Z 2.550} C_DIS
   LIN {X -0.892, Y 21.127, Z 2.550} C_DIS
   LIN {X -0.892, Y 21.586, Z 2.550} C_DIS
   LIN {X -0.897, Y 22.112, Z 2.550} C_DIS
   LIN {X -0.904, Y 22.595, Z 2.550} C_DIS
   LIN {X -0.917, Y 23.123, Z 2.550} C_DIS
   LIN {X -0.930, Y 23.602, Z 2.550} C_DIS
   LIN {X -0.950, Y 24.129, Z 2.550} C_DIS
   LIN {X -0.971, Y 24.633, Z 2.550} C_DIS
   LIN {X -0.997, Y 25.145, Z 2.550} C_DIS
   LIN {X -1.023, Y 25.616, Z 2.550} C_DIS
   LIN {X -1.055, Y 26.112, Z 2.550} C_DIS
   LIN {X -1.090, Y 26.605, Z 2.550} C_DIS
   LIN {X -1.129, Y 27.113, Z 2.550} C_DIS
   LIN {X -1.172, Y 27.627, Z 2.550} C_DIS
   LIN {X -1.219, Y 28.132, Z 2.550} C_DIS
   LIN {X -1.268, Y 28.639, Z 2.550} C_DIS
   LIN {X -1.320, Y 29.127, Z 2.550} C_DIS
   LIN {X -1.376, Y 29.627, Z 2.550} C_DIS
   LIN {X -1.434, Y 30.110, Z 2.550} C_DIS
   LIN {X -1.499, Y 30.628, Z 2.550} C_DIS
   LIN {X -1.563, Y 31.106, Z 2.550} C_DIS
   LIN {X -1.634, Y 31.614, Z 2.550} C_DIS
   LIN {X -1.703, Y 32.086, Z 2.550} C_DIS
   LIN {X -1.784, Y 32.609, Z 2.550} C_DIS
   LIN {X -1.861, Y 33.085, Z 2.550} C_DIS
   LIN {X -1.951, Y 33.621, Z 2.550} C_DIS
   LIN {X -2.030, Y 34.070, Z 2.550} C_DIS
   LIN {X -2.133, Y 34.634, Z 2.550} C_DIS
   LIN {X -2.213, Y 35.048, Z 2.550} C_DIS
   LIN {X -2.325, Y 35.621, Z 2.550} C_DIS
   LIN {X -2.446, Y 36.221, Z 2.550} C_DIS
   LIN {X -2.524, Y 36.611, Z 2.550} C_DIS
   LIN {X -2.573, Y 36.930, Z 2.550} C_DIS
   LIN {X -2.620, Y 37.380, Z 2.550} C_DIS
   LIN {X -2.611, Y 37.692, Z 2.550} C_DIS
   LIN {X -2.567, Y 38.084, Z 2.550} C_DIS
   LIN {X -2.409, Y 38.718, Z 2.550} C_DIS
   LIN {X -2.279, Y 39.062, Z 2.550} C_DIS
   LIN {X -1.989, Y 39.603, Z 2.550} C_DIS
   LIN {X -1.774, Y 39.901, Z 2.550} C_DIS
   LIN {X -1.269, Y 40.438, Z 2.550} C_DIS
   LIN {X -0.978, Y 40.670, Z 2.550} C_DIS
   LIN {X -0.480, Y 40.985, Z 2.550} C_DIS
   LIN {X -0.111, Y 41.150, Z 2.550} C_DIS
   LIN {X 0.441, Y 41.330, Z 2.550} C_DIS
   LIN {X 0.814, Y 41.389, Z 2.550} C_DIS
   LIN {X 1.514, Y 41.426, Z 2.550} C_DIS
   LIN {X 1.890, Y 41.379, Z 2.550} C_DIS
   LIN {X 2.474, Y 41.261, Z 2.550} C_DIS
   LIN {X 2.943, Y 41.082, Z 2.550} C_DIS
   LIN {X 3.305, Y 40.912, Z 2.550} C_DIS
   LIN {X 3.800, Y 40.574, Z 2.550} C_DIS
   LIN {X 4.057, Y 40.366, Z 2.550} C_DIS
   LIN {X 4.510, Y 39.858, Z 2.550} C_DIS
   LIN {X 4.685, Y 39.627, Z 2.550} C_DIS
   LIN {X 5.054, Y 38.859, Z 2.550} C_DIS
   LIN {X 5.216, Y 38.465, Z 2.550} C_DIS
   LIN {X 5.360, Y 37.931, Z 2.550} C_DIS
   LIN {X 5.457, Y 37.569, Z 2.550} C_DIS
   LIN {X 5.558, Y 37.177, Z 2.550} C_DIS
   LIN {X 5.822, Y 36.149, Z 2.550} C_DIS
   LIN {X 5.869, Y 35.961, Z 2.550} C_DIS
   LIN {X 6.062, Y 35.173, Z 2.550} C_DIS
   LIN {X 6.109, Y 34.976, Z 2.550} C_DIS
   LIN {X 6.290, Y 34.207, Z 2.550} C_DIS
   LIN {X 6.334, Y 34.016, Z 2.550} C_DIS
   LIN {X 6.509, Y 33.241, Z 2.550} C_DIS
   LIN {X 6.557, Y 33.025, Z 2.550} C_DIS
   LIN {X 6.723, Y 32.259, Z 2.550} C_DIS
   LIN {X 6.768, Y 32.043, Z 2.550} C_DIS
   LIN {X 6.924, Y 31.291, Z 2.550} C_DIS
   LIN {X 6.967, Y 31.078, Z 2.550} C_DIS
   LIN {X 7.122, Y 30.294, Z 2.550} C_DIS
   LIN {X 7.167, Y 30.059, Z 2.550} C_DIS
   LIN {X 7.315, Y 29.272, Z 2.550} C_DIS
   LIN {X 7.357, Y 29.043, Z 2.550} C_DIS
   LIN {X 7.490, Y 28.301, Z 2.550} C_DIS
   LIN {X 7.528, Y 28.079, Z 2.550} C_DIS
   LIN {X 7.654, Y 27.335, Z 2.550} C_DIS
   LIN {X 7.694, Y 27.091, Z 2.550} C_DIS
   LIN {X 7.814, Y 26.344, Z 2.550} C_DIS
   LIN {X 7.850, Y 26.108, Z 2.550} C_DIS
   LIN {X 7.963, Y 25.364, Z 2.550} C_DIS
   LIN {X 8.002, Y 25.094, Z 2.550} C_DIS
   LIN {X 8.107, Y 24.348, Z 2.550} C_DIS
   LIN {X 8.141, Y 24.097, Z 2.550} C_DIS
   LIN {X 8.238, Y 23.369, Z 2.550} C_DIS
   LIN {X 8.271, Y 23.110, Z 2.550} C_DIS
   LIN {X 8.361, Y 22.380, Z 2.550}
   LaserEnd_Ext()
   LIN {X -13.280, Y -25.489, Z 2.550}
   LaserStart_Ext()
   LIN {X -13.280, Y -22.131, Z 2.550}
   LaserEnd_Ext()
   LIN {X -12.280, Y -19.648, Z 2.550}
   LaserStart_Ext()
   LIN {X -12.280, Y -27.993, Z 2.550}
   LaserEnd_Ext()
   LIN {X -11.280, Y -29.285, Z 2.550}
   LaserStart_Ext()
   LIN {X -11.280, Y -18.076, Z 2.550}
   LaserEnd_Ext()
   LIN {X -10.280, Y -16.447, Z 2.550}
   LaserStart_Ext()
   LIN {X -10.280, Y -30.173, Z 2.550}
   LaserEnd_Ext()
   LIN {X -9.280, Y -30.812, Z 2.550}
   LaserStart_Ext()
   LIN {X -9.280, Y -14.718, Z 2.550}
   LaserEnd_Ext()
   LIN {X -8.280, Y -12.871, Z 2.550}
   LaserStart_Ext()
   LIN {X -8.280, Y -31.271, Z 2.550}
   LaserEnd_Ext()
   LIN {X -7.280, Y -31.565, Z 2.550}
   LaserStart_Ext()
   LIN {X -7.280, Y -10.887, Z 2.550}
   LaserEnd_Ext()
   LIN {X -6.280, Y -8.739, Z 2.550}
   LaserStart_Ext()
   LIN {X -6.280, Y -31.723, Z 2.550}
   LaserEnd_Ext()
   LIN {X -5.280, Y -31.757, Z 2.550}
   LaserStart_Ext()
   LIN {X -5.280, Y -6.395, Z 2.550}
   LaserEnd_Ext()
   LIN {X -4.280, Y -3.791, Z 2.550}
   LaserStart_Ext()
   LIN {X -4.280, Y -31.666, Z 2.550}
   LaserEnd_Ext()
   LIN {X -3.280, Y -31.448, Z 2.550}
   LaserStart_Ext()
   LIN {X -3.280, Y -0.840, Z 2.550}
   LaserEnd_Ext()
   LIN {X -2.280, Y 2.631, Z 2.550}
   LaserStart_Ext()
   LIN {X -2.280, Y -31.089, Z 2.550}
   LaserEnd_Ext()
   LIN {X -1.280, Y -30.563, Z 2.550}
   LaserStart_Ext()
   LIN {X -1.280, Y 6.992, Z 2.550}
   LaserEnd_Ext()
   LIN {X -1.280, Y 35.488, Z 2.550}
   LaserStart_Ext()
   LIN {X -1.280, Y 38.809, Z 2.550}
   LaserEnd_Ext()
   LIN {X -0.280, Y 39.929, Z 2.550}
   LaserStart_Ext()
   LIN {X -0.280, Y 28.803, Z 2.550}
   LaserEnd_Ext()
   LIN {X -0.280, Y 13.669, Z 2.550}
   LaserStart_Ext()
   LIN {X -0.280, Y -29.836, Z 2.550}
   LaserEnd_Ext()
   LIN {X 0.720, Y -28.818, Z 2.550}
   LaserStart_Ext()
   LIN {X 0.720, Y 40.362, Z 2.550}
   LaserEnd_Ext()
   LIN {X 1.720, Y 40.392, Z 2.550}
   LaserStart_Ext()
   LIN {X 1.720, Y -27.271, Z 2.550}
   LaserEnd_Ext()
   LIN {X 2.720, Y -24.565, Z 2.550}
   LaserStart_Ext()
   LIN {X 2.720, Y 40.082, Z 2.550}
   LaserEnd_Ext()
   LIN {X 3.720, Y 39.241, Z 2.550}
   LaserStart_Ext()
   LIN {X 3.720, Y -21.345, Z 2.550}
   LaserEnd_Ext()
   LIN {X 4.720, Y -17.711, Z 2.550}
   LaserStart_Ext()
   LIN {X 4.720, Y 36.419, Z 2.550}
   LaserEnd_Ext()
   LIN {X 5.720, Y 32.165, Z 2.550}
   LaserStart_Ext()
   LIN {X 5.720, Y -13.465, Z 2.550}
   LaserEnd_Ext()
   LIN {X 6.720, Y -8.170, Z 2.550}
   LaserStart_Ext()
   LIN {X 6.720, Y 26.847, Z 2.550}
   LaserEnd_Ext()
   LIN {X 7.720, Y 18.860, Z 2.550}
   LaserStart_Ext()
   LIN {X 7.720, Y -0.214, Z 2.550}
   LaserEnd_Ext()
   LIN {X 8.969, Y 3.104, Z 3.400}
   LaserStart_Ext()
   LIN {X 8.939, Y 2.595, Z 3.400} C_DIS
   LIN {X 8.908, Y 2.086, Z 3.400} C_DIS
   LIN {X 8.873, Y 1.569, Z 3.400} C_DIS
   LIN {X 8.838, Y 1.070, Z 3.400} C_DIS
   LIN {X 8.798, Y 0.555, Z 3.400} C_DIS
   LIN {X 8.758, Y 0.060, Z 3.400} C_DIS
   LIN {X 8.714, Y -0.451, Z 3.400} C_DIS
   LIN {X 8.671, Y -0.933, Z 3.400} C_DIS
   LIN {X 8.623, Y -1.439, Z 3.400} C_DIS
   LIN {X 8.577, Y -1.910, Z 3.400} C_DIS
   LIN {X 8.523, Y -2.426, Z 3.400} C_DIS
   LIN {X 8.480, Y -2.831, Z 3.400} C_DIS
   LIN {X 8.404, Y -3.494, Z 3.400} C_DIS
   LIN {X 8.365, Y -3.832, Z 3.400} C_DIS
   LIN {X 8.284, Y -4.485, Z 3.400} C_DIS
   LIN {X 8.243, Y -4.815, Z 3.400} C_DIS
   LIN {X 8.155, Y -5.479, Z 3.400} C_DIS
   LIN {X 8.111, Y -5.808, Z 3.400} C_DIS
   LIN {X 8.019, Y -6.460, Z 3.400} C_DIS
   LIN {X 7.973, Y -6.781, Z 3.400} C_DIS
   LIN {X 7.873, Y -7.442, Z 3.400} C_DIS
   LIN {X 7.821, Y -7.780, Z 3.400} C_DIS
   LIN {X 7.718, Y -8.425, Z 3.400} C_DIS
   LIN {X 7.659, Y -8.786, Z 3.400} C_DIS
   LIN {X 7.553, Y -9.412, Z 3.400} C_DIS
   LIN {X 7.493, Y -9.761, Z 3.400} C_DIS
   LIN {X 7.383, Y -10.375, Z 3.400} C_DIS
   LIN {X 7.318, Y -10.737, Z 3.400} C_DIS
   LIN {X 7.186, Y -11.436, Z 3.400} C_DIS
   LIN {X 7.127, Y -11.746, Z 3.400} C_DIS
   LIN {X 7.003, Y -12.373, Z 3.400} C_DIS
   LIN {X 6.907, Y -12.849, Z 3.400} C_DIS
   LIN {X 6.793, Y -13.396, Z 3.400} C_DIS
   LIN {X 6.711, Y -13.789, Z 3.400} C_DIS
   LIN {X 6.574, Y -14.415, Z 3.400} C_DIS
   LIN {X 6.503, Y -14.743, Z 3.400} C_DIS
   LIN {X 6.347, Y -15.428, Z 3.400} C_DIS
   LIN {X 6.277, Y -15.734, Z 3.400} C_DIS
   LIN {X 6.113, Y -16.426, Z 3.400} C_DIS
   LIN {X 6.042, Y -16.721, Z 3.400} C_DIS
   LIN {X 5.875, Y -17.397, Z 3.400} C_DIS
   LIN {X 5.786, Y -17.753, Z 3.400} C_DIS
   LIN {X 5.641, Y -18.321, Z 3.400} C_DIS
   LIN {X 5.534, Y -18.732, Z 3.400} C_DIS
   LIN {X 5.383, Y -19.301, Z 3.400} C_DIS
   LIN {X 5.276, Y -19.699, Z 3.400} C_DIS
   LIN {X 5.122, Y -20.257, Z 3.400} C_DIS
   LIN {X 5.011, Y -20.654, Z 3.400} C_DIS
   LIN {X 4.850, Y -21.219, Z 3.400} C_DIS
   LIN {X 4.734, Y -21.618, Z 3.400} C_DIS
   LIN {X 4.565, Y -22.191, Z 3.400} C_DIS
   LIN {X 4.475, Y -22.493, Z 3.400} C_DIS
   LIN {X 4.299, Y -23.068, Z 3.400} C_DIS
   LIN {X 4.212, Y -23.353, Z 3.400} C_DIS
   LIN {X 3.919, Y -24.282, Z 3.400} C_DIS
   LIN {X 3.540, Y -25.449, Z 3.400} C_DIS
   LIN {X 3.478, Y -25.634, Z 3.400} C_DIS
   LIN {X 3.273, Y -26.242, Z 3.400} C_DIS
   LIN {X 3.158, Y -26.587, Z 3.400} C_DIS
   LIN {X 3.044, Y -26.844, Z 3.400} C_DIS
   LIN {X 2.745, Y -27.578, Z 3.400} C_DIS
   LIN {X 2.559, Y -27.852, Z 3.400} C_DIS
   LIN {X 1.824, Y -29.088, Z 3.400} C_DIS
   LIN {X 1.430, Y -29.581, Z 3.400} C_DIS
   LIN {X 1.176, Y -29.857, Z 3.400} C_DIS
   LIN {X 0.749, Y -30.288, Z 3.400} C_DIS
   LIN {X 0.429, Y -30.567, Z 3.400} C_DIS
   LIN {X 0.032, Y -30.890, Z 3.400} C_DIS
   LIN {X -0.366, Y -31.170, Z 3.400} C_DIS
   LIN {X -0.784, Y -31.440, Z 3.400} C_DIS
   LIN {X -1.224, Y -31.682, Z 3.400} C_DIS
   LIN {X -1.645, Y -31.893, Z 3.400} C_DIS
   LIN {X -2.125, Y -32.093, Z 3.400} C_DIS
   LIN {X -2.546, Y -32.250, Z 3.400} C_DIS
   LIN {X -3.069, Y -32.405, Z 3.400} C_DIS
   LIN {X -3.491, Y -32.513, Z 3.400} C_DIS
   LIN {X -4.032, Y -32.612, Z 3.400} C_DIS
   LIN {X -4.436, Y -32.670, Z 3.400} C_DIS
   LIN {X -5.000, Y -32.712, Z 3.400} C_DIS
   LIN {X -5.392, Y -32.725, Z 3.400} C_DIS
   LIN {X -5.986, Y -32.704, Z 3.400} C_DIS
   LIN {X -6.368, Y -32.675, Z 3.400} C_DIS
   LIN {X -6.969, Y -32.589, Z 3.400} C_DIS
   LIN {X -7.332, Y -32.521, Z 3.400} C_DIS
   LIN {X -7.914, Y -32.372, Z 3.400} C_DIS
   LIN {X -8.250, Y -32.272, Z 3.400} C_DIS
   LIN {X -8.839, Y -32.053, Z 3.400} C_DIS
   LIN {X -9.150, Y -31.921, Z 3.400} C_DIS
   LIN {X -9.722, Y -31.634, Z 3.400} C_DIS
   LIN {X -10.014, Y -31.469, Z 3.400} C_DIS
   LIN {X -10.548, Y -31.123, Z 3.400} C_DIS
   LIN {X -10.820, Y -30.928, Z 3.400} C_DIS
   LIN {X -11.320, Y -30.522, Z 3.400} C_DIS
   LIN {X -11.561, Y -30.306, Z 3.400} C_DIS
   LIN {X -12.017, Y -29.846, Z 3.400} C_DIS
   LIN {X -12.233, Y -29.605, Z 3.400} C_DIS
   LIN {X -12.637, Y -29.098, Z 3.400} C_DIS
   LIN {X -12.822, Y -28.838, Z 3.400} C_DIS
   LIN {X -13.180, Y -28.270, Z 3.400} C_DIS
   LIN {X -13.330, Y -27.999, Z 3.400} C_DIS
   LIN {X -13.622, Y -27.400, Z 3.400} C_DIS
   LIN {X -13.743, Y -27.113, Z 3.400} C_DIS
   LIN {X -13.961, Y -26.508, Z 3.400} C_DIS
   LIN {X -14.050, Y -26.209, Z 3.400} C_DIS
   LIN {X -14.206, Y -25.571, Z 3.400} C_DIS
   LIN {X -14.263, Y -25.259, Z 3.400} C_DIS
   LIN {X -14.348, Y -24.617, Z 3.400} C_DIS
   LIN {X -14.371, Y -24.294, Z 3.400} C_DIS
   LIN {X -14.386, Y -23.660, Z 3.400} C_DIS
   LIN {X -14.373, Y -23.320, Z 3.400} C_DIS
   LIN {X -14.321, Y -22.698, Z 3.400} C_DIS
   LIN {X -14.271, Y -22.355, Z 3.400} C_DIS
   LIN {X -14.191, Y -21.908, Z 3.400} C_DIS
   LIN {X -14.067, Y -21.426, Z 3.400} C_DIS
   LIN {X -13.972, Y -21.071, Z 3.400} C_DIS
   LIN {X -13.512, Y -19.953, Z 3.400} C_DIS
   LIN {X -13.387, Y -19.647, Z 3.400} C_DIS
   LIN {X -12.972, Y -18.936, Z 3.400} C_DIS
   LIN {X -12.895, Y -18.802, Z 3.400} C_DIS
   LIN {X -12.618, Y -18.371, Z 3.400} C_DIS
   LIN {X -12.171, Y -17.683, Z 3.400} C_DIS
   LIN {X -12.034, Y -17.468, Z 3.400} C_DIS
   LIN {X -11.877, Y -17.213, Z 3.400} C_DIS
   LIN {X -10.910, Y -15.591, Z 3.400} C_DIS
   LIN {X -10.685, Y -15.220, Z 3.400} C_DIS
   LIN {X -10.461, Y -14.838, Z 3.400} C_DIS
   LIN {X -10.237, Y -14.443, Z 3.400} C_DIS
   LIN {X -9.962, Y -13.950, Z 3.400} C_DIS
   LIN {X -9.744, Y -13.552, Z 3.400} C_DIS
   LIN {X -9.479, Y -13.060, Z 3.400} C_DIS
   LIN {X -9.264, Y -12.654, Z 3.400} C_DIS
   LIN {X -9.008, Y -12.162, Z 3.400} C_DIS
   LIN {X -8.797, Y -11.752, Z 3.400} C_DIS
   LIN {X -8.552, Y -11.263, Z 3.400} C_DIS
   LIN {X -8.347, Y -10.851, Z 3.400} C_DIS
   LIN {X -8.114, Y -10.369, Z 3.400} C_DIS
   LIN {X -7.917, Y -9.958, Z 3.400} C_DIS
   LIN {X -7.692, Y -9.479, Z 3.400} C_DIS
   LIN {X -7.498, Y -9.058, Z 3.400} C_DIS
   LIN {X -7.280, Y -8.577, Z 3.400} C_DIS
   LIN {X -7.089, Y -8.149, Z 3.400} C_DIS
   LIN {X -6.880, Y -7.667, Z 3.400} C_DIS
   LIN {X -6.693, Y -7.232, Z 3.400} C_DIS
   LIN {X -6.488, Y -6.743, Z 3.400} C_DIS
   LIN {X -6.301, Y -6.290, Z 3.400} C_DIS
   LIN {X -6.101, Y -5.795, Z 3.400} C_DIS
   LIN {X -5.920, Y -5.337, Z 3.400} C_DIS
   LIN {X -5.734, Y -4.856, Z 3.400} C_DIS
   LIN {X -5.564, Y -4.411, Z 3.400} C_DIS
   LIN {X -5.389, Y -3.938, Z 3.400} C_DIS
   LIN {X -5.226, Y -3.492, Z 3.400} C_DIS
   LIN {X -5.058, Y -3.020, Z 3.400} C_DIS
   LIN {X -4.896, Y -2.558, Z 3.400} C_DIS
   LIN {X -4.732, Y -2.076, Z 3.400} C_DIS
   LIN {X -4.572, Y -1.598, Z 3.400} C_DIS
   LIN {X -4.268, Y -0.650, Z 3.400} C_DIS
   LIN {X -4.171, Y -0.346, Z 3.400} C_DIS
   LIN {X -4.078, Y -0.043, Z 3.400} C_DIS
   LIN {X -3.884, Y 0.602, Z 3.400} C_DIS
   LIN {X -3.675, Y 1.325, Z 3.400} C_DIS
   LIN {X -3.568, Y 1.711, Z 3.400} C_DIS
   LIN {X -3.377, Y 2.405, Z 3.400} C_DIS
   LIN {X -3.291, Y 2.732, Z 3.400} C_DIS
   LIN {X -3.162, Y 3.232, Z 3.400} C_DIS
   LIN {X -3.043, Y 3.706, Z 3.400} C_DIS
   LIN {X -2.918, Y 4.218, Z 3.400} C_DIS
   LIN {X -2.805, Y 4.698, Z 3.400} C_DIS
   LIN {X -2.683, Y 5.228, Z 3.400} C_DIS
   LIN {X -2.580, Y 5.699, Z 3.400} C_DIS
   LIN {X -2.470, Y 6.209, Z 3.400} C_DIS
   LIN {X -2.377, Y 6.665, Z 3.400} C_DIS
   LIN {X -2.274, Y 7.177, Z 3.400} C_DIS
   LIN {X -2.193, Y 7.601, Z 3.400} C_DIS
   LIN {X -2.079, Y 8.216, Z 3.400} C_DIS
   LIN {X -2.016, Y 8.573, Z 3.400} C_DIS
   LIN {X -1.901, Y 9.243, Z 3.400} C_DIS
   LIN {X -1.849, Y 9.569, Z 3.400} C_DIS
   LIN {X -1.744, Y 10.234, Z 3.400} C_DIS
   LIN {X -1.696, Y 10.566, Z 3.400} C_DIS
   LIN {X -1.604, Y 11.210, Z 3.400} C_DIS
   LIN {X -1.556, Y 11.566, Z 3.400} C_DIS
   LIN {X -1.478, Y 12.177, Z 3.400} C_DIS
   LIN {X -1.434, Y 12.548, Z 3.400} C_DIS
   LIN {X -1.361, Y 13.175, Z 3.400} C_DIS
   LIN {X -1.323, Y 13.543, Z 3.400} C_DIS
   LIN {X -1.258, Y 14.189, Z 3.400} C_DIS
   LIN {X -1.223, Y 14.573, Z 3.400} C_DIS
   LIN {X -1.170, Y 15.180, Z 3.400} C_DIS
   LIN {X -1.138, Y 15.598, Z 3.400} C_DIS
   LIN {X -1.097, Y 16.162, Z 3.400} C_DIS
   LIN {X -1.070, Y 16.584, Z 3.400} C_DIS
   LIN {X -1.037, Y 17.144, Z 3.400} C_DIS
   LIN {X -1.016, Y 17.569, Z 3.400} C_DIS
   LIN {X -0.990, Y 18.143, Z 3.400} C_DIS
   LIN {X -0.975, Y 18.568, Z 3.400} C_DIS
   LIN {X -0.956, Y 19.157, Z 3.400} C_DIS
   LIN {X -0.947, Y 19.578, Z 3.400} C_DIS
   LIN {X -0.936, Y 20.161, Z 3.400} C_DIS
   LIN {X -0.933, Y 20.575, Z 3.400} C_DIS
   LIN {X -0.931, Y 21.152, Z 3.400} C_DIS
   LIN {X -0.933, Y 21.556, Z 3.400} C_DIS
   LIN {X -0.938, Y 22.145, Z 3.400} C_DIS
   LIN {X -0.946, Y 22.553, Z 3.400} C_DIS
   LIN {X -0.960, Y 23.153, Z 3.400} C_DIS
   LIN {X -0.973, Y 23.561, Z 3.400} C_DIS
   LIN {X -0.995, Y 24.171, Z 3.400} C_DIS
   LIN {X -1.014, Y 24.573, Z 3.400} C_DIS
   LIN {X -1.045, Y 25.175, Z 3.400} C_DIS
   LIN {X -1.068, Y 25.565, Z 3.400} C_DIS
   LIN {X -1.106, Y 26.159, Z 3.400} C_DIS
   LIN {X -1.135, Y 26.551, Z 3.400} C_DIS
   LIN {X -1.184, Y 27.169, Z 3.400} C_DIS
   LIN {X -1.218, Y 27.557, Z 3.400} C_DIS
   LIN {X -1.275, Y 28.181, Z 3.400} C_DIS
   LIN {X -1.314, Y 28.561, Z 3.400} C_DIS
   LIN {X -1.379, Y 29.174, Z 3.400} C_DIS
   LIN {X -1.422, Y 29.550, Z 3.400} C_DIS
   LIN {X -1.496, Y 30.168, Z 3.400} C_DIS
   LIN {X -1.545, Y 30.543, Z 3.400} C_DIS
   LIN {X -1.628, Y 31.163, Z 3.400} C_DIS
   LIN {X -1.678, Y 31.515, Z 3.400} C_DIS
   LIN {X -1.775, Y 32.170, Z 3.400} C_DIS
   LIN {X -1.825, Y 32.488, Z 3.400} C_DIS
   LIN {X -1.939, Y 33.186, Z 3.400} C_DIS
   LIN {X -1.989, Y 33.477, Z 3.400} C_DIS
   LIN {X -2.105, Y 34.132, Z 3.400} C_DIS
   LIN {X -2.161, Y 34.440, Z 3.400} C_DIS
   LIN {X -2.264, Y 34.980, Z 3.400} C_DIS
   LIN {X -2.350, Y 35.418, Z 3.400} C_DIS
   LIN {X -2.478, Y 36.053, Z 3.400} C_DIS
   LIN {X -2.601, Y 36.661, Z 3.400} C_DIS
   LIN {X -2.664, Y 37.467, Z 3.400} C_DIS
   LIN {X -2.694, Y 37.764, Z 3.400} C_DIS
   LIN {X -2.649, Y 38.096, Z 3.400} C_DIS
   LIN {X -2.580, Y 38.494, Z 3.400} C_DIS
   LIN {X -2.332, Y 39.159, Z 3.400} C_DIS
   LIN {X -2.193, Y 39.467, Z 3.400} C_DIS
   LIN {X -1.700, Y 40.141, Z 3.400} C_DIS
   LIN {X -1.574, Y 40.292, Z 3.400} C_DIS
   LIN {X -1.333, Y 40.477, Z 3.400} C_DIS
   LIN {X -0.755, Y 40.941, Z 3.400} C_DIS
   LIN {X -0.249, Y 41.167, Z 3.400} C_DIS
   LIN {X 0.184, Y 41.348, Z 3.400} C_DIS
   LIN {X 1.104, Y 41.477, Z 3.400} C_DIS
   LIN {X 1.222, Y 41.493, Z 3.400} C_DIS
   LIN {X 1.361, Y 41.475, Z 3.400} C_DIS
   LIN {X 2.184, Y 41.380, Z 3.400} C_DIS
   LIN {X 2.402, Y 41.306, Z 3.400} C_DIS
   LIN {X 3.060, Y 41.062, Z 3.400} C_DIS
   LIN {X 3.532, Y 40.757, Z 3.400} C_DIS
   LIN {X 3.861, Y 40.533, Z 3.400} C_DIS
   LIN {X 4.280, Y 40.085, Z 3.400} C_DIS
   LIN {X 4.510, Y 39.828, Z 3.400} C_DIS
   LIN {X 4.778, Y 39.263, Z 3.400} C_DIS
   LIN {X 5.135, Y 38.531, Z 3.400} C_DIS
   LIN {X 5.286, Y 37.971, Z 3.400} C_DIS
   LIN {X 5.432, Y 37.430, Z 3.400} C_DIS
   LIN {X 5.646, Y 36.593, Z 3.400} C_DIS
   LIN {X 5.868, Y 35.733, Z 3.400} C_DIS
   LIN {X 5.955, Y 35.378, Z 3.400} C_DIS
   LIN {X 6.103, Y 34.766, Z 3.400} C_DIS
   LIN {X 6.186, Y 34.414, Z 3.400} C_DIS
   LIN {X 6.330, Y 33.798, Z 3.400} C_DIS
   LIN {X 6.413, Y 33.432, Z 3.400} C_DIS
   LIN {X 6.550, Y 32.820, Z 3.400} C_DIS
   LIN {X 6.631, Y 32.444, Z 3.400} C_DIS
   LIN {X 6.760, Y 31.844, Z 3.400} C_DIS
   LIN {X 6.838, Y 31.466, Z 3.400} C_DIS
   LIN {X 6.961, Y 30.868, Z 3.400} C_DIS
   LIN {X 7.037, Y 30.482, Z 3.400} C_DIS
   LIN {X 7.159, Y 29.860, Z 3.400} C_DIS
   LIN {X 7.233, Y 29.465, Z 3.400} C_DIS
   LIN {X 7.346, Y 28.859, Z 3.400} C_DIS
   LIN {X 7.413, Y 28.480, Z 3.400} C_DIS
   LIN {X 7.517, Y 27.892, Z 3.400} C_DIS
   LIN {X 7.583, Y 27.505, Z 3.400} C_DIS
   LIN {X 7.682, Y 26.916, Z 3.400} C_DIS
   LIN {X 7.745, Y 26.520, Z 3.400} C_DIS
   LIN {X 7.838, Y 25.936, Z 3.400} C_DIS
   LIN {X 7.899, Y 25.527, Z 3.400} C_DIS
   LIN {X 7.987, Y 24.939, Z 3.400} C_DIS
   LIN {X 8.046, Y 24.524, Z 3.400} C_DIS
   LIN {X 8.128, Y 23.933, Z 3.400} C_DIS
   LIN {X 8.182, Y 23.527, Z 3.400} C_DIS
   LIN {X 8.258, Y 22.947, Z 3.400} C_DIS
   LIN {X 8.309, Y 22.533, Z 3.400} C_DIS
   LIN {X 8.377, Y 21.970, Z 3.400} C_DIS
   LIN {X 8.424, Y 21.561, Z 3.400} C_DIS
   LIN {X 8.489, Y 20.984, Z 3.400} C_DIS
   LIN {X 8.532, Y 20.571, Z 3.400} C_DIS
   LIN {X 8.590, Y 20.014, Z 3.400} C_DIS
   LIN {X 8.632, Y 19.577, Z 3.400} C_DIS
   LIN {X 8.686, Y 19.005, Z 3.400} C_DIS
   LIN {X 8.723, Y 18.575, Z 3.400} C_DIS
   LIN {X 8.765, Y 18.094, Z 3.400} C_DIS
   LIN {X 8.812, Y 17.494, Z 3.400} C_DIS
   LIN {X 8.848, Y 17.012, Z 3.400} C_DIS
   LIN {X 8.879, Y 16.566, Z 3.400} C_DIS
   LIN {X 8.915, Y 16.014, Z 3.400} C_DIS
   LIN {X 8.942, Y 15.575, Z 3.400} C_DIS
   LIN {X 8.973, Y 15.032, Z 3.400} C_DIS
   LIN {X 8.996, Y 14.587, Z 3.400} C_DIS
   LIN {X 9.022, Y 14.044, Z 3.400} C_DIS
   LIN {X 9.041, Y 13.591, Z 3.400} C_DIS
   LIN {X 9.063, Y 13.043, Z 3.400} C_DIS
   LIN {X 9.078, Y 12.579, Z 3.400} C_DIS
   LIN {X 9.094, Y 12.046, Z 3.400} C_DIS
   LIN {X 9.105, Y 11.571, Z 3.400} C_DIS
   LIN {X 9.116, Y 11.044, Z 3.400} C_DIS
   LIN {X 9.123, Y 10.584, Z 3.400} C_DIS
   LIN {X 9.129, Y 10.063, Z 3.400} C_DIS
   LIN {X 9.132, Y 9.598, Z 3.400} C_DIS
   LIN {X 9.134, Y 9.081, Z 3.400} C_DIS
   LIN {X 9.132, Y 8.605, Z 3.400} C_DIS
   LIN {X 9.129, Y 8.096, Z 3.400} C_DIS
   LIN {X 9.123, Y 7.602, Z 3.400} C_DIS
   LIN {X 9.115, Y 7.081, Z 3.400} C_DIS
   LIN {X 9.104, Y 6.569, Z 3.400} C_DIS
   LIN {X 9.091, Y 6.063, Z 3.400} C_DIS
   LIN {X 9.076, Y 5.563, Z 3.400} C_DIS
   LIN {X 9.059, Y 5.071, Z 3.400} C_DIS
   LIN {X 9.040, Y 4.584, Z 3.400} C_DIS
   LIN {X 9.019, Y 4.092, Z 3.400} C_DIS
   LIN {X 8.995, Y 3.605, Z 3.400} C_DIS
   LIN {X 8.969, Y 3.104, Z 3.400}
   LaserEnd_Ext()
   LIN {X -7.808, Y -31.360, Z 3.400}
   LaserStart_Ext()
   LIN {X -3.062, Y -31.360, Z 3.400}
   LaserEnd_Ext()
   LIN {X -0.955, Y -30.360, Z 3.400}
   LaserStart_Ext()
   LIN {X -9.887, Y -30.360, Z 3.400}
   LaserEnd_Ext()
   LIN {X -11.091, Y -29.360, Z 3.400}
   LaserStart_Ext()
   LIN {X 0.261, Y -29.360, Z 3.400}
   LaserEnd_Ext()
   LIN {X 1.093, Y -28.360, Z 3.400}
   LaserStart_Ext()
   LIN {X -11.935, Y -28.360, Z 3.400}
   LaserEnd_Ext()
   LIN {X -12.529, Y -27.360, Z 3.400}
   LaserStart_Ext()
   LIN {X 1.689, Y -27.360, Z 3.400}
   LaserEnd_Ext()
   LIN {X 2.165, Y -26.360, Z 3.400}
   LaserStart_Ext()
   LIN {X -12.951, Y -26.360, Z 3.400}
   LaserEnd_Ext()
   LIN {X -13.228, Y -25.360, Z 3.400}
   LaserStart_Ext()
   LIN {X 2.515, Y -25.360, Z 3.400}
   LaserEnd_Ext()
   LIN {X 2.842, Y -24.360, Z 3.400}
   LaserStart_Ext()
   LIN {X -13.364, Y -24.360, Z 3.400}
   LaserEnd_Ext()
   LIN {X -13.373, Y -23.360, Z 3.400}
   LaserStart_Ext()
   LIN {X 3.162, Y -23.360, Z 3.400}
   LaserEnd_Ext()
   LIN {X 3.470, Y -22.360, Z 3.400}
   LaserStart_Ext()
   LIN {X -13.256, Y -22.360, Z 3.400}
   LaserEnd_Ext()
   LIN {X -13.010, Y -21.360, Z 3.400}
   LaserStart_Ext()
   LIN {X 3.768, Y -21.360, Z 3.400}
   LaserEnd_Ext()
   LIN {X 4.055, Y -20.360, Z 3.400}
   LaserStart_Ext()
   LIN {X -12.598, Y -20.360, Z 3.400}
   LaserEnd_Ext()
   LIN {X -12.062, Y -19.360, Z 3.400}
   LaserStart_Ext()
   LIN {X 4.331, Y -19.360, Z 3.400}
   LaserEnd_Ext()
   LIN {X 4.598, Y -18.360, Z 3.400}
   LaserStart_Ext()
   LIN {X -11.418, Y -18.360, Z 3.400}
   LaserEnd_Ext()
   LIN {X -10.801, Y -17.360, Z 3.400}
   LaserStart_Ext()
   LIN {X 4.854, Y -17.360, Z 3.400}
   LaserEnd_Ext()
   LIN {X 5.100, Y -16.360, Z 3.400}
   LaserStart_Ext()
   LIN {X -10.204, Y -16.360, Z 3.400}
   LaserEnd_Ext()
   LIN {X -9.608, Y -15.360, Z 3.400}
   LaserStart_Ext()
   LIN {X 5.336, Y -15.360, Z 3.400}
   LaserEnd_Ext()
   LIN {X 5.563, Y -14.360, Z 3.400}
   LaserStart_Ext()
   LIN {X -9.047, Y -14.360, Z 3.400}
   LaserEnd_Ext()
   LIN {X -8.506, Y -13.360, Z 3.400}
   LaserStart_Ext()
   LIN {X 5.779, Y -13.360, Z 3.400}
   LaserEnd_Ext()
   LIN {X 5.985, Y -12.360, Z 3.400}
   LaserStart_Ext()
   LIN {X -7.986, Y -12.360, Z 3.400}
   LaserEnd_Ext()
   LIN {X -7.484, Y -11.360, Z 3.400}
   LaserStart_Ext()
   LIN {X 6.182, Y -11.360, Z 3.400}
   LaserEnd_Ext()
   LIN {X 6.370, Y -10.360, Z 3.400}
   LaserStart_Ext()
   LIN {X -7.001, Y -10.360, Z 3.400}
   LaserEnd_Ext()
   LIN {X -6.537, Y -9.360, Z 3.400}
   LaserStart_Ext()
   LIN {X 6.547, Y -9.360, Z 3.400}
   LaserEnd_Ext()
   LIN {X 6.715, Y -8.360, Z 3.400}
   LaserStart_Ext()
   LIN {X -6.091, Y -8.360, Z 3.400}
   LaserEnd_Ext()
   LIN {X -5.662, Y -7.360, Z 3.400}
   LaserStart_Ext()
   LIN {X 6.874, Y -7.360, Z 3.400}
   LaserEnd_Ext()
   LIN {X 7.023, Y -6.360, Z 3.400}
   LaserStart_Ext()
   LIN {X -5.251, Y -6.360, Z 3.400}
   LaserEnd_Ext()
   LIN {X -4.857, Y -5.360, Z 3.400}
   LaserStart_Ext()
   LIN {X 7.162, Y -5.360, Z 3.400}
   LaserEnd_Ext()
   LIN {X 7.292, Y -4.360, Z 3.400}
   LaserStart_Ext()
   LIN {X -4.479, Y -4.360, Z 3.400}
   LaserEnd_Ext()
   LIN {X -4.117, Y -3.360, Z 3.400}
   LaserStart_Ext()
   LIN {X 7.413, Y -3.360, Z 3.400}
   LaserEnd_Ext()
   LIN {X 7.524, Y -2.360, Z 3.400}
   LaserStart_Ext()
   LIN {X -3.772, Y -2.360, Z 3.400}
   LaserEnd_Ext()
   LIN {X -3.445, Y -1.360, Z 3.400}
   LaserStart_Ext()
   LIN {X 7.626, Y -1.360, Z 3.400}
   LaserEnd_Ext()
   LIN {X 7.718, Y -0.360, Z 3.400}
   LaserStart_Ext()
   LIN {X -3.130, Y -0.360, Z 3.400}
   LaserEnd_Ext()
   LIN {X -2.832, Y 0.640, Z 3.400}
   LaserStart_Ext()
   LIN {X 7.801, Y 0.640, Z 3.400}
   LaserEnd_Ext()
   LIN {X 7.875, Y 1.640, Z 3.400}
   LaserStart_Ext()
   LIN {X -2.550, Y 1.640, Z 3.400}
   LaserEnd_Ext()
   LIN {X -2.282, Y 2.640, Z 3.400}
   LaserStart_Ext()
   LIN {X 7.940, Y 2.640, Z 3.400}
   LaserEnd_Ext()
   LIN {X 7.995, Y 3.640, Z 3.400}
   LaserStart_Ext()
   LIN {X -2.030, Y 3.640, Z 3.400}
   LaserEnd_Ext()
   LIN {X -1.792, Y 4.640, Z 3.400}
   LaserStart_Ext()
   LIN {X 8.041, Y 4.640, Z 3.400}
   LaserEnd_Ext()
   LIN {X 8.078, Y 5.640, Z 3.400}
   LaserStart_Ext()
   LIN {X -1.570, Y 5.640, Z 3.400}
   LaserEnd_Ext()
   LIN {X -1.362, Y 6.640, Z 3.400}
   LaserStart_Ext()
   LIN {X 8.105, Y 6.640, Z 3.400}
   LaserEnd_Ext()
   LIN {X 8.123, Y 7.640, Z 3.400}
   LaserStart_Ext()
   LIN {X -1.169, Y 7.640, Z 3.400}
   LaserEnd_Ext()
   LIN {X -0.990, Y 8.640, Z 3.400}
   LaserStart_Ext()
   LIN {X 8.132, Y 8.640, Z 3.400}
   LaserEnd_Ext()
   LIN {X 8.132, Y 9.640, Z 3.400}
   LaserStart_Ext()
   LIN {X -0.825, Y 9.640, Z 3.400}
   LaserEnd_Ext()
   LIN {X -0.675, Y 10.640, Z 3.400}
   LaserStart_Ext()
   LIN {X 8.122, Y 10.640, Z 3.400}
   LaserEnd_Ext()
   LIN {X 8.103, Y 11.640, Z 3.400}
   LaserStart_Ext()
   LIN {X -0.539, Y 11.640, Z 3.400}
   LaserEnd_Ext()
   LIN {X -0.416, Y 12.640, Z 3.400}
   LaserStart_Ext()
   LIN {X 8.075, Y 12.640, Z 3.400}
   LaserEnd_Ext()
   LIN {X 8.038, Y 13.640, Z 3.400}
   LaserStart_Ext()
   LIN {X -0.308, Y 13.640, Z 3.400}
   LaserEnd_Ext()
   LIN {X -0.213, Y 14.640, Z 3.400}
   LaserStart_Ext()
   LIN {X 7.992, Y 14.640, Z 3.400}
   LaserEnd_Ext()
   LIN {X 7.936, Y 15.640, Z 3.400}
   LaserStart_Ext()
   LIN {X -0.133, Y 15.640, Z 3.400}
   LaserEnd_Ext()
   LIN {X -0.065, Y 16.640, Z 3.400}
   LaserStart_Ext()
   LIN {X 7.871, Y 16.640, Z 3.400}
   LaserEnd_Ext()
   LIN {X 7.797, Y 17.640, Z 3.400}
   LaserStart_Ext()
   LIN {X -0.012, Y 17.640, Z 3.400}
   LaserEnd_Ext()
   LIN {X 0.028, Y 18.640, Z 3.400}
   LaserStart_Ext()
   LIN {X 7.714, Y 18.640, Z 3.400}
   LaserEnd_Ext()
   LIN {X 7.621, Y 19.640, Z 3.400}
   LaserStart_Ext()
   LIN {X 0.054, Y 19.640, Z 3.400}
   LaserEnd_Ext()
   LIN {X 0.067, Y 20.640, Z 3.400}
   LaserStart_Ext()
   LIN {X 7.519, Y 20.640, Z 3.400}
   LaserEnd_Ext()
   LIN {X 7.408, Y 21.640, Z 3.400}
   LaserStart_Ext()
   LIN {X 0.067, Y 21.640, Z 3.400}
   LaserEnd_Ext()
   LIN {X 0.053, Y 22.640, Z 3.400}
   LaserStart_Ext()
   LIN {X 7.288, Y 22.640, Z 3.400}
   LaserEnd_Ext()
   LIN {X 7.158, Y 23.640, Z 3.400}
   LaserStart_Ext()
   LIN {X 0.025, Y 23.640, Z 3.400}
   LaserEnd_Ext()
   LIN {X -0.016, Y 24.640, Z 3.400}
   LaserStart_Ext()
   LIN {X 7.019, Y 24.640, Z 3.400}
   LaserEnd_Ext()
   LIN {X 6.871, Y 25.640, Z 3.400}
   LaserStart_Ext()
   LIN {X -0.071, Y 25.640, Z 3.400}
   LaserEnd_Ext()
   LIN {X -0.139, Y 26.640, Z 3.400}
   LaserStart_Ext()
   LIN {X 6.713, Y 26.640, Z 3.400}
   LaserEnd_Ext()
   LIN {X 6.546, Y 27.640, Z 3.400}
   LaserStart_Ext()
   LIN {X -0.221, Y 27.640, Z 3.400}
   LaserEnd_Ext()
   LIN {X -0.317, Y 28.640, Z 3.400}
   LaserStart_Ext()
   LIN {X 6.369, Y 28.640, Z 3.400}
   LaserEnd_Ext()
   LIN {X 6.183, Y 29.640, Z 3.400}
   LaserStart_Ext()
   LIN {X -0.426, Y 29.640, Z 3.400}
   LaserEnd_Ext()
   LIN {X -0.549, Y 30.640, Z 3.400}
   LaserStart_Ext()
   LIN {X 5.987, Y 30.640, Z 3.400}
   LaserEnd_Ext()
   LIN {X 5.781, Y 31.640, Z 3.400}
   LaserStart_Ext()
   LIN {X -0.686, Y 31.640, Z 3.400}
   LaserEnd_Ext()
   LIN {X -0.837, Y 32.640, Z 3.400}
   LaserStart_Ext()
   LIN {X 5.565, Y 32.640, Z 3.400}
   LaserEnd_Ext()
   LIN {X 5.340, Y 33.640, Z 3.400}
   LaserStart_Ext()
   LIN {X -1.002, Y 33.640, Z 3.400}
   LaserEnd_Ext()
   LIN {X -1.181, Y 34.640, Z 3.400}
   LaserStart_Ext()
   LIN {X 5.105, Y 34.640, Z 3.400}
   LaserEnd_Ext()
   LIN {X 4.859, Y 35.640, Z 3.400}
   LaserStart_Ext()
   LIN {X -1.375, Y 35.640, Z 3.400}
   LaserEnd_Ext()
   LIN {X -1.576, Y 36.640, Z 3.400}
   LaserStart_Ext()
   LIN {X 4.602, Y 36.640, Z 3.400}
   LaserEnd_Ext()
   LIN {X 4.339, Y 37.640, Z 3.400}
   LaserStart_Ext()
   LIN {X -1.676, Y 37.640, Z 3.400}
   LaserEnd_Ext()
   LIN {X -1.459, Y 38.640, Z 3.400}
   LaserStart_Ext()
   LIN {X 3.969, Y 38.640, Z 3.400}
   LaserEnd_Ext()
   LIN {X 3.327, Y 39.640, Z 3.400}
   LaserStart_Ext()
   LIN {X -0.781, Y 39.640, Z 3.400}
   LaserEnd_Ext()
   LIN {X -11.955, Y -29.789, Z 4.250}
   LaserStart_Ext()
   LIN {X -12.160, Y -29.557, Z 4.250} C_DIS
   LIN {X -12.561, Y -29.055, Z 4.250} C_DIS
   LIN {X -12.742, Y -28.799, Z 4.250} C_DIS
   LIN {X -13.093, Y -28.243, Z 4.250} C_DIS
   LIN {X -13.256, Y -27.952, Z 4.250} C_DIS
   LIN {X -13.539, Y -27.370, Z 4.250} C_DIS
   LIN {X -13.663, Y -27.077, Z 4.250} C_DIS
   LIN {X -13.874, Y -26.490, Z 4.250} C_DIS
   LIN {X -13.969, Y -26.179, Z 4.250} C_DIS
   LIN {X -14.122, Y -25.555, Z 4.250} C_DIS
   LIN {X -14.180, Y -25.258, Z 4.250} C_DIS
   LIN {X -14.264, Y -24.618, Z 4.250} C_DIS
   LIN {X -14.286, Y -24.397, Z 4.250} C_DIS
   LIN {X -14.183, Y -23.679, Z 4.250} C_DIS
   LIN {X -14.008, Y -21.987, Z 4.250} C_DIS
   LIN {X -14.013, Y -21.468, Z 4.250} C_DIS
   LIN {X -13.901, Y -21.051, Z 4.250} C_DIS
   LIN {X -13.819, Y -20.850, Z 4.250} C_DIS
   LIN {X -13.319, Y -19.626, Z 4.250} C_DIS
   LIN {X -13.152, Y -19.340, Z 4.250} C_DIS
   LIN {X -12.830, Y -18.780, Z 4.250} C_DIS
   LIN {X -12.337, Y -18.014, Z 4.250} C_DIS
   LIN {X -11.983, Y -17.456, Z 4.250} C_DIS
   LIN {X -10.560, Y -15.072, Z 4.250} C_DIS
   LIN {X -10.306, Y -14.636, Z 4.250} C_DIS
   LIN {X -10.028, Y -14.117, Z 4.250} C_DIS
   LIN {X -9.655, Y -13.445, Z 4.250} C_DIS
   LIN {X -9.290, Y -12.767, Z 4.250} C_DIS
   LIN {X -8.933, Y -12.081, Z 4.250} C_DIS
   LIN {X -8.826, Y -11.868, Z 4.250} C_DIS
   LIN {X -8.480, Y -11.179, Z 4.250} C_DIS
   LIN {X -8.378, Y -10.971, Z 4.250} C_DIS
   LIN {X -8.045, Y -10.284, Z 4.250} C_DIS
   LIN {X -7.946, Y -10.074, Z 4.250} C_DIS
   LIN {X -7.622, Y -9.384, Z 4.250} C_DIS
   LIN {X -7.529, Y -9.178, Z 4.250} C_DIS
   LIN {X -7.212, Y -8.477, Z 4.250} C_DIS
   LIN {X -7.121, Y -8.270, Z 4.250} C_DIS
   LIN {X -6.813, Y -7.561, Z 4.250} C_DIS
   LIN {X -6.726, Y -7.357, Z 4.250} C_DIS
   LIN {X -6.422, Y -6.630, Z 4.250} C_DIS
   LIN {X -6.337, Y -6.421, Z 4.250} C_DIS
   LIN {X -6.038, Y -5.678, Z 4.250} C_DIS
   LIN {X -5.958, Y -5.474, Z 4.250} C_DIS
   LIN {X -5.676, Y -4.744, Z 4.250} C_DIS
   LIN {X -5.602, Y -4.545, Z 4.250} C_DIS
   LIN {X -5.333, Y -3.821, Z 4.250} C_DIS
   LIN {X -5.262, Y -3.624, Z 4.250} C_DIS
   LIN {X -5.003, Y -2.893, Z 4.250} C_DIS
   LIN {X -4.934, Y -2.694, Z 4.250} C_DIS
   LIN {X -4.678, Y -1.940, Z 4.250} C_DIS
   LIN {X -4.556, Y -1.565, Z 4.250} C_DIS
   LIN {X -4.198, Y -0.448, Z 4.250} C_DIS
   LIN {X -3.928, Y 0.452, Z 4.250} C_DIS
   LIN {X -3.856, Y 0.693, Z 4.250} C_DIS
   LIN {X -3.815, Y 0.832, Z 4.250} C_DIS
   LIN {X -3.421, Y 2.248, Z 4.250} C_DIS
   LIN {X -3.205, Y 3.075, Z 4.250} C_DIS
   LIN {X -3.008, Y 3.866, Z 4.250} C_DIS
   LIN {X -2.963, Y 4.054, Z 4.250} C_DIS
   LIN {X -2.773, Y 4.866, Z 4.250} C_DIS
   LIN {X -2.731, Y 5.052, Z 4.250} C_DIS
   LIN {X -2.554, Y 5.858, Z 4.250} C_DIS
   LIN {X -2.516, Y 6.037, Z 4.250} C_DIS
   LIN {X -2.354, Y 6.827, Z 4.250} C_DIS
